	//
	//	List of READ (and WRITE) commands.
	// NOTE: Monitoring loop stops on first cmd = ''.
	//
	cmdList_Read_HIPACE30:	ARRAY [1..16] OF T_CRYO_PUMP_CMD := [
		(cmd := cfg.C_CMD_bON, 				length := 20),	// 20 chars with the terminator!	
		(cmd := cfg.C_CMD_nCtrlMode, 		length := 17),	
		(cmd := cfg.C_CMD_sErrorCode, 		length := 20),
		(cmd := cfg.C_CMD_bTargetSpeed, 	length := 20),
		(cmd := cfg.C_CMD_nMotorCurr, 		length := 20),
		(cmd := cfg.C_CMD_nPumpHours, 		length := 20),
		(cmd := cfg.C_CMD_nMotorVolt, 		length := 20),
		(cmd := cfg.C_CMD_nElecHours, 		length := 20),
		(cmd := cfg.C_CMD_nElecTemp, 		length := 20),
		(cmd := cfg.C_CMD_nPumpTemp, 		length := 20),
		(cmd := cfg.C_CMD_nPumpSpeed, 		length := 20),
		(cmd := '', 						length := 0),
		(cmd := '', 						length := 0),
		(cmd := '', 						length := 0),
		(cmd := '', 						length := 0),
		(cmd := '', 						length := 0)];
	
		i:	INT;
END_VAR
IF NOT bStarted	THEN
	//
	// START: Mandatory for ALL pumps !!!
	//
	// Set references from FB_RS_BASE
	cfgRef	REF=cfg;
	ctrlRef	REF=ctrl;
	statRef	REF=stat;

	// Set references from FB_CRYO_TMP_BASE
	cfgBaseRef	REF=cfg;
	ctrlBaseRef	REF=ctrl;
	statBaseRef	REF=stat;
	
	// Copy input parameters to configuration
	cfg.nModel			:= in_nModel;
	cfg.bAutoMonitor	:= in_bAutoMonitor;
	cfg.tDelay_Periodic	:= DINT_TO_TIME(in_nPeriod);
	
	
	// Set pointers to arrays of commands
	ptrInitCmds	:= ADR(cfg.cmdList_Init);(* Pointer to INIT commands *)
	ptrReadCmds	:= ADR(cfg.cmdList_Read);(* Pointer to READ commands *)
	
	// TODO in FB that extends the functionality
	// Set pointers to comm, i.e.
	ptrCommCfg	:= ADR(comm.cfg);	(* Pointer to comm.cfg instance *)
	ptrCommCtrl	:= ADR(comm.ctrl);	(* Pointer to comm.ctrl instance *)
	ptrCommStat	:= ADR(comm.stat);	(* Pointer to comm.stat instance *)
	
	// Set comm suffixes for commands and replies
	ptrCommCfg^.sCmdSuffix		:= in_sCmdSuffix;
	ptrCommCfg^.sReplySuffix	:= in_sReplySuffix;

	statRef.bConfigured	:= TRUE;
	bStarted			:= TRUE;
	//
	// END: Mandatory for ALL pumps !!!
	//


	//
	// ATH specific configuration
	//
	
	// Assign INIT and READ commands.
	cfg.cmdList_Init	:= cmdList_Init_HIPACE30;
	cfg.cmdList_Read	:= cmdList_Read_HIPACE30;
	
	// Add checksum to all INIT and READ commands
	FOR i:=1 TO 8 DO
		IF cfg.cmdList_Init[i].cmd <> '' THEN
			cfg.cmdList_Init[i].cmd	:= M_PVP_Checksum(cfg.cmdList_Init[i].cmd);
		ELSE
			EXIT;
		END_IF
	END_FOR
	
	FOR i:=1 TO 16 DO
		IF cfg.cmdList_Read[i].cmd <> '' THEN
			cfg.cmdList_Read[i].cmd	:= M_PVP_Checksum(cfg.cmdList_Read[i].cmd);
		ELSE
			EXIT;
		END_IF
	END_FOR
	
END_IF
END_METHOD

METHOD M_GetSpeed : DINT
VAR_INPUT
END_VAR
M_GetSpeed	:= stat.nPumpSpeed;
END_METHOD

METHOD M_IsReady : BOOL
VAR_INPUT
END_VAR
M_IsReady	:= stat.bReady;
END_METHOD

METHOD M_IsRunning : BOOL
VAR_INPUT
END_VAR
M_IsRunning	:= stat.bMoving;
END_METHOD

METHOD M_ReadFromReply : BOOL
// Method to check correctness of the reply and assign the result to a status variable.
VAR_INPUT
	idx:		INT;		(* arr [idx] will hold the first extracted value, arr [idx+1] the second one, etc. *)
	bInitCmd:	BOOL := FALSE;
END_VAR
VAR
	pos:	INT;
	cmd:	STRING;
	length:	DINT;
	subStr:	STRING;
	valLen:	INT;		// Number of character for the value
END_VAR
// During INIT it might happen that the command index is 0.
// These cases should be discarded.
IF idx <= 0	THEN
	M_ReadFromReply	:= TRUE;
	RETURN;
END_IF

IF bInitCmd	THEN
	cmd		:= cfg.cmdList_Init[idx].cmd;
	length	:= cfg.cmdList_Init[idx].length;
ELSE
	cmd		:= cfg.cmdList_Read[idx].cmd;
	length	:= cfg.cmdList_Read[idx].length;
END_IF

IF length <> 0  AND  LEN(stat.sReply) <> length THEN
	stat.sErrorText	:= 'Wrong reply length';
	M_ReadFromReply	:= FALSE;
	RETURN;
END_IF

// Check if sent command was correct.
IF	FIND(stat.sReply,'NO_DEF') > 0	OR 
	FIND(stat.sReply,'_RANGE') > 0	OR 
	FIND(stat.sReply,'_LOGIC') > 0		THEN
	// Wrong command sent. This is an error.
	stat.sErrorText	:= 'Incorrect command';
	M_ReadFromReply	:= FALSE;
	RETURN;
END_IF

// Check the structure of the reply.
// Example 1 - Data query with 6 characters for the value:
//    CMD:   1 2 3 0 0 3 0 9 0 2 = ? 1 1 2 cR
//    Reply: 1 2 3 1 0 3 0 9 0 6 0 0 0 6 3 3 0 3 7 cR
//    valLen = 6 (from '06' in reply)
//    value = 633
// Example 2 - Data query with 3 characters for the value:
//    CMD:   1 2 3 0 0 0 6 0 0 2 = ? x x x cR
//    Reply: 1 2 3 1 0 0 6 0 0 3 0 0 2 y y y cR
//    valLen = 3 (from '03' in reply)
//    value = 002 = 2
// Example 3 - Command (reply is identical to command):
//    CMD:   0 4 2 1 0 0 1 0 0 6 1 1 1 1 1 1 0 2 0 cR
//    Reply: 0 4 2 1 0 0 1 0 0 6 1 1 1 1 1 1 0 2 0 cR
//    valLen = 6 (from '06' in reply)
//    value = 111111
//
// Compared to the first 10 chars of the command, 
// the reply should modify characters 3 and 9 (index starts from 0)
// reply[3] = 1
// reply[9] = length - 14
//
// So, we want to convert: 1 2 3 0 0 3 0 9 0 2
//                     to: 1 2 3 1 0 3 0 9 0 6
// Extract first 10 characters from the command
subStr	:= MID(cmd,10,1);
// Replace character [3] with '1', i.e. with ASCII 49.
subStr[3]	:= 49;
// Replace character [9] with expected number of characters in the value.
valLen	:= DINT_TO_INT(length - 14);
// Convert integer to character.
subStr[9]	:= INT_TO_BYTE(valLen + 48);	// 48 is ascii '0'.
IF	FIND(stat.sReply,subStr) <> 1	THEN
	// Wrong reply received. This is an error.
	stat.sErrorText	:= 'Wrong reply received';
	M_ReadFromReply	:= FALSE;
	RETURN;
END_IF


//
// All fine so far. Let's extract the reading.
//
// The actual reply is contained in the 'valLen' (3 or 6) characters starting 
// from char [10] (11-the character for MID() function).
subStr	:= MID(stat.sReply, valLen, 11);

// Remove the 3-character checksum from the command.
cmd	:= MID(cmd, LEN(cmd)-3,1);


IF cmd = cfg.C_CMD_sFwVersion	THEN
	stat.sFwVersion		:= MID(subStr, 6, 1);
ELSIF cmd = cfg.C_CMD_sHwVersion	THEN
	stat.sHwVersion		:= MID(subStr, 6, 1);
ELSIF cmd = cfg.C_CMD_nNominalSpeed	THEN
	stat.nNominalSpeed	:= LREAL_TO_DINT(STRING_TO_LREAL(subStr));
ELSIF cmd = cfg.C_CMD_bON	THEN
	stat.bON	:= STRING_TO_BOOL(subStr) <> FALSE;
ELSIF cmd = cfg.C_CMD_nCtrlMode	THEN
	stat.nCtrlMode	:= STRING_TO_DINT(subStr);
ELSIF cmd = cfg.C_CMD_sErrorCode	THEN
	IF	FIND(subStr,'Err') > 0	OR 
		FIND(subStr,'Wrn') > 0		THEN
		// There is an Error or Warning.
		stat.sFailureCode	:= MID(subStr, 6, 1);
		stat.bFailure		:= TRUE;
	ELSE
		stat.sFailureCode	:= 'OK';
		stat.bFailure		:= FALSE;
	END_IF
ELSIF cmd = cfg.C_CMD_bTargetSpeed	THEN
	stat.bTargetSpeed	:= STRING_TO_BOOL(subStr) <> FALSE;
ELSIF cmd = cfg.C_CMD_nMotorCurr	THEN
	stat.nMotorCurr	:= STRING_TO_DINT(subStr) * 10;	// [mA]
ELSIF cmd = cfg.C_CMD_nPumpHours	THEN
	stat.nPumpHours	:= STRING_TO_DINT(subStr);
ELSIF cmd = cfg.C_CMD_nMotorVolt	THEN
	stat.nMotorVolt	:= STRING_TO_DINT(subStr) / 100;
	stat.lrMotorVolt:= STRING_TO_LREAL(subStr) / 100.0;	// [V]
ELSIF cmd = cfg.C_CMD_nElecHours	THEN
	stat.nElecHours	:= STRING_TO_DINT(subStr);
ELSIF cmd = cfg.C_CMD_nElecTemp	THEN
	stat.nElecTemp	:= STRING_TO_DINT(subStr);
ELSIF cmd = cfg.C_CMD_nPumpTemp	THEN
	stat.nPumpTemp	:= STRING_TO_DINT(subStr);
ELSIF cmd = cfg.C_CMD_nPumpSpeed	THEN
	stat.nPumpSpeed	:= LREAL_TO_DINT(STRING_TO_LREAL(subStr));
END_IF


M_ReadFromReply	:= TRUE;	// OK
END_METHOD

METHOD M_UpdateStatus
VAR_INPUT
END_VAR
// Update Status from digital inputs readings
stat.bReady		:= i_bReady;
stat.bFailure	:= NOT i_bError;	// Active low

stat.bMoving	:= stat.bReady OR stat.nPumpSpeed > 0;

// Set Control Mode Label
(*
	1 = remote
	2 = RS-485
	4 = PV.can
	8 = Fieldbus
	16 = E74
	255 = unlock interface selection
*)
CASE stat.nCtrlMode	OF
	1:		stat.sCtrlMode	:= 'REMOTE';
	2:		stat.sCtrlMode	:= 'RS-485';
	4:		stat.sCtrlMode	:= 'PV.can';
	8:		stat.sCtrlMode	:= 'FIELDBUS';
	16:		stat.sCtrlMode	:= 'E74';
ELSE
	stat.sCtrlMode	:= 'UNKNOWN';
END_CASE
END_METHOD

END_FUNCTION_BLOCK

// ---- POUs/Subsystems/Examples/Evacuation/FB_CRYO_EVAC_ECODRY_ATH2303M.TcPOU
FUNCTION_BLOCK FB_CRYO_EVAC_ECODRY_ATH2303M EXTENDS FB_CRYO_EVAC_BASE
VAR_INPUT
END_VAR
VAR_OUTPUT
END_VAR
VAR
	rp:	FB_CRYO_PUMP_ECODRY;	// Roughing Pump
	tp:	FB_CRYO_PUMP_ATH2303M;	// Turbo Molecular Pump
	
END_VAR

SUPER^();

METHOD M_Configure
VAR_INPUT
END_VAR
//
// Specific PDS IR Imager configuration.
//
IF NOT stat.bConfigured	THEN
	// MANDATORY: Set References !!!
	// If not done, system will crash !!!
	rpRef	REF=rp;
	tpRef	REF=tp;
	

	// Specific instance configuration, e.g. anything different
	// from the default values given in the cfg structure of type T_CRYO_EVAC_CFG.
	cfg.nPressGaugeType1	:= E_CRYO_SENSOR_TYPE_PRESS.WRG_D_NW25;
	cfg.nPressGaugeType2	:= E_CRYO_SENSOR_TYPE_PRESS.PKR_360;

	cfg.lrThld_Prevac := 5.0;	// Prevacuum pressure threshold
	// Cryo pressure threshold to start Turbo Pump before opening Valve
	cfg.lrThld_TP_SafeStartPressure := 0.01;	
	// Cryo pressure threshold to start Turbo Pump once Valve is open
	cfg.lrThld_Valve_SafeOpenPressure := 0.1;	
	cfg.tDelay := T#3S;	// Time delay before stopping Turbo Pump

	stat.bConfigured	:= TRUE;;
ELSE
	RETURN;	// Nothing to do any more
END_IF
END_METHOD

METHOD M_ExecuteControllers
VAR_INPUT
END_VAR
//
// Specific Cryo Lab Evacuation System HW configuration.
//

// Roughing Pump	
rp(	
	in_bSimulation	:= FALSE,
	in_sName		:= 'ECODRY V01',
	in_bEnable		:= ctrl.bEnable_RP,
	in_nSlaveID		:= 31,
	in_sVersion		:= 'V01',
	in_nPeriod		:= 2000);

// Turbo Molecular Pump
tp(	
	in_bSimulation	:= FALSE,
	in_sName		:= 'ATH2303M',
	in_bEnable		:= ctrl.bEnable_TP,
	in_nModel		:= 2303,
	in_bAutoMonitor	:= TRUE,
	in_nPeriod		:= 2000);

// Valve
valve(
	in_bEnable		:= ctrl.bEnable_Valve,
	in_nFeedback	:= E_CRYO_BIN_ACT_FEEDBACK.ON_AND_OFF);
END_METHOD

END_FUNCTION_BLOCK

// ---- POUs/Pumps/FB_CRYO_PUMP_ECODRY.TcPOU
FUNCTION_BLOCK FB_CRYO_PUMP_ECODRY EXTENDS FB_CRYO_PUMP_MODBUS
VAR_INPUT
END_VAR
VAR_OUTPUT
END_VAR
VAR CONSTANT
END_VAR
VAR
	{attribute 'OPC.UA.DA' := '1'}
	cfg:		T_CRYO_PUMP_MODBUS_CFG;		//  Config parameters
	{attribute 'OPC.UA.DA' := '1'}
	ctrl:		T_CRYO_PUMP_MODBUS_CTRL;	//  Control parameters
	{attribute 'OPC.UA.DA' := '1'}
	{attribute 'OPC.UA.DA.Access' := '1'}
	stat:		T_CRYO_PUMP_MODBUS_STAT;	//  Status parameters - ReadOnly


END_VAR

// Execute the base class object FB_RS_BASE
SUPER^();

METHOD M_Configure
VAR_INPUT
END_VAR
IF NOT bStarted	THEN
	//
	// START: Mandatory for ALL pumps !!!
	//
	// Set references from FB_RS_BASE
	cfgRef	REF=cfg;
	ctrlRef	REF=ctrl;
	statRef	REF=stat;

	// Set references from FB_CRYO_PUMP_BASE
	cfgBaseRef	REF=cfg;
	ctrlBaseRef	REF=ctrl;
	statBaseRef	REF=stat;

	// Set references from FB_CRYO_PUMP_MODBUS
	cfgModbusRef	REF=cfg;
	ctrlModbusRef	REF=ctrl;
	statModbusRef	REF=stat;

	// Copy input parameters to configuration
	cfg.nModel			:= in_nModel;
	cfg.bAutoMonitor	:= in_bAutoMonitor;
	cfg.tDelay_Periodic	:= DINT_TO_TIME(in_nPeriod);
	
	
	// Set pointers to arrays of commands
//	ptrInitCmds	:= ADR(cfg.cmdList_Init);(* Pointer to INIT commands *)
//	ptrReadCmds	:= ADR(cfg.cmdList_Read);(* Pointer to READ commands *)
	
	// TODO in FB that extends the functionality
	// Set pointers to comm, i.e.
	ptrCommCfg	:= ADR(comm.cfg);	(* Pointer to comm.cfg instance *)
	ptrCommCtrl	:= ADR(comm.ctrl);	(* Pointer to comm.ctrl instance *)
	ptrCommStat	:= ADR(comm.stat);	(* Pointer to comm.stat instance *)
	
	// Set comm suffixes for commands and replies
//	ptrCommCfg^.sCmdSuffix		:= '';
//	ptrCommCfg^.sReplySuffix	:= '';

	statRef.bConfigured	:= TRUE;
	bStarted			:= TRUE;
	//
	// END: Mandatory for ALL pumps !!!
	//


	// TODO USER
	// Add here real configuration
	IF in_sVersion = 'V01'	THEN
		cfg.nVersion	:= E_ECODRY_VERSION.V01;
	ELSIF in_sVersion = 'V21'  OR  in_sVersion = 'V22'	THEN
		cfg.nVersion	:= E_ECODRY_VERSION.V21_22;
	END_IF
	
	// Adjust addresses and number of words
	CASE cfg.nVersion	OF
		E_ECODRY_VERSION.V01:
			// Set register addresses
			cfg.aAddr [1]	:= 16#0040;
			cfg.aAddr [2]	:= 16#0067;
			cfg.aAddr [3]	:= 16#0667;
			cfg.aAddr [4]	:= 0;	// Unused address must be zero
			
			// Set number of words to read
			cfg.aWords [1]	:= 16;
			cfg.aWords [2]	:= 2;
			cfg.aWords [3]	:= 6;
			cfg.aWords [4]	:= 0;	// Number of words for unused address must be zero
	END_CASE
	
	cfg.nSlaveID	:= in_nSlaveID;

	
END_IF
END_METHOD

METHOD M_ExtractReadings_V01 : BOOL
VAR_INPUT
	nAddressIndex:	INT;	// Which address space to read
END_VAR
VAR
	pBuf:	POINTER TO BYTE	:= ADR(stat.nInputBuffer);
	loop:	INT;
	par:	INT;
END_VAR
// There are 3 bytes before data starts !!!
IF nAddressIndex = 1 THEN
	////////////////////////////
	// Extract Common Parameters
	////////////////////////////

	// Reference Frequency 0x40H
	// Offset 3 + 0 = 3
	stat.lrFreqRef		:= UINT_TO_LREAL(M_ByteSwapUINT(ADR(pBuf[3]))) / 100.0;
	stat.lrOutFreq		:= INT_TO_LREAL(M_ByteSwapINT(ADR(pBuf[5]))) / 100.0;
	stat.nPumpSpeed		:= LREAL_TO_DINT(stat.lrOutFreq * 60.0);	// [Hz] -> [rpm]
	stat.nMotorCurr		:= UINT_TO_DINT(M_ByteSwapUINT(ADR(pBuf[7]))) * 10;
	stat.lrOutVoltRef	:= UINT_TO_LREAL(M_ByteSwapUINT(ADR(pBuf[13]))) / 10.0;
	stat.nMotorVolt		:= UINT_TO_DINT(M_ByteSwapUINT(ADR(pBuf[15])));
	stat.lrOutPower		:= INT_TO_LREAL(M_ByteSwapINT(ADR(pBuf[17]))) / 10.0;
	
	stat.nOpTime	:= M_ByteSwapUINT(ADR(pBuf[27]));
	stat.nSwFlash	:= M_ByteSwapUINT(ADR(pBuf[29]));

	(*
	stat.lrTemperature	:= UINT_TO_LREAL(M_ByteSwapUINT(ADR(pBuf[83])));

	stat.nSwRom		:= M_ByteSwapUINT(ADR(pBuf[57]));
	stat.nNumRunCmd	:= M_ByteSwapUINT(ADR(pBuf[109]));
	stat.nFanOpTime	:= M_ByteSwapUINT(ADR(pBuf[81]));
	*)

ELSIF nAddressIndex = 2 THEN
	stat.nFanOpTime			:= M_ByteSwapUINT(ADR(pBuf[3]));
	stat.nElecTemp			:= UINT_TO_DINT(M_ByteSwapUINT(ADR(pBuf[5])));
ELSIF nAddressIndex = 3 THEN
	stat.nServiceHours		:= M_ByteSwapUINT(ADR(pBuf[3]));
	stat.nNumPumpDowns		:= M_ByteSwapUINT(ADR(pBuf[7]));
	stat.nDaysUntilService	:= M_ByteSwapUINT(ADR(pBuf[13]));
END_IF
END_METHOD

METHOD M_ExtractReadings_V21_22 : BOOL
VAR_INPUT
	nAddressIndex:	INT;	// Which address space to read
END_VAR
VAR
	pBuf:	POINTER TO BYTE	:= ADR(stat.nInputBuffer);
	loop:	INT;
	par:	INT;
END_VAR
// There are 3 bytes before data starts !!!
IF nAddressIndex = 1 THEN
	////////////////////////////
	// Extract Common Parameters
	////////////////////////////

	// Reference Frequency 0x40H
	// Offset 3 + 0 = 3
	stat.lrFreqRef		:= UINT_TO_LREAL(M_ByteSwapUINT(ADR(pBuf[3]))) / 100.0;
	stat.lrOutFreq		:= INT_TO_LREAL(M_ByteSwapINT(ADR(pBuf[5]))) / 100.0;
	stat.nMotorCurr		:= UINT_TO_DINT(M_ByteSwapUINT(ADR(pBuf[7]))) * 10;
	stat.lrOutVoltRef	:= UINT_TO_LREAL(M_ByteSwapUINT(ADR(pBuf[13]))) / 10.0;
	stat.nMotorVolt		:= UINT_TO_DINT(M_ByteSwapUINT(ADR(pBuf[15])));
	stat.lrOutPower		:= INT_TO_LREAL(M_ByteSwapINT(ADR(pBuf[17]))) / 10.0;
	
	stat.nOpTime	:= M_ByteSwapUINT(ADR(pBuf[27]));
	stat.nSwFlash	:= M_ByteSwapUINT(ADR(pBuf[29]));

	(*
	stat.lrTemperature	:= UINT_TO_LREAL(M_ByteSwapUINT(ADR(pBuf[83])));

	stat.nSwRom		:= M_ByteSwapUINT(ADR(pBuf[57]));
	stat.nNumRunCmd	:= M_ByteSwapUINT(ADR(pBuf[109]));
	stat.nFanOpTime	:= M_ByteSwapUINT(ADR(pBuf[81]));
	*)

ELSIF nAddressIndex = 2 THEN
	stat.nFanOpTime			:= M_ByteSwapUINT(ADR(pBuf[3]));
	stat.nElecTemp			:= UINT_TO_DINT(M_ByteSwapUINT(ADR(pBuf[5])));
ELSIF nAddressIndex = 3 THEN
	stat.nServiceHours		:= M_ByteSwapUINT(ADR(pBuf[3]));
	stat.nNumPumpDowns		:= M_ByteSwapUINT(ADR(pBuf[7]));
	stat.nDaysUntilService	:= M_ByteSwapUINT(ADR(pBuf[13]));
END_IF
END_METHOD

METHOD M_IsReady : BOOL
VAR_INPUT
END_VAR
//	M_UpdateStatus() sets the stat.bReady flag.
M_IsReady	:= stat.bReady;
END_METHOD

METHOD M_IsRunning : BOOL
VAR_INPUT
END_VAR
M_IsRunning	:= stat.bReady OR stat.nPumpSpeed > 0;
END_METHOD

METHOD M_ReadFromReply : BOOL
VAR_INPUT
	nAddressIndex:	INT;	// Which address space to read
END_VAR
IF cfg.nVersion	= E_ECODRY_VERSION.V01	THEN
	M_ExtractReadings_V01    (nAddressIndex);
ELSIF cfg.nVersion	= E_ECODRY_VERSION.V21_22	THEN
	M_ExtractReadings_V21_22 (nAddressIndex);
END_IF
END_METHOD

METHOD M_UpdateStatus
VAR_INPUT
END_VAR
// Update inputs
stat.bReady		:= NOT i_bRunning;	// Active low
END_METHOD

END_FUNCTION_BLOCK

// ---- POUs/Pumps/FB_CRYO_PUMP_MODBUS.TcPOU
FUNCTION_BLOCK FB_CRYO_PUMP_MODBUS EXTENDS FB_CRYO_PUMP_BASE
VAR_INPUT
	{attribute 'OPC.UA.DA' := '0'}
	in_nSlaveID:	BYTE := 1;		// Slave ID
	{attribute 'OPC.UA.DA' := '0'}
	in_sVersion:	STRING := 'V21';	// Version number. String starting with 'V', e.g. 'V21'.
END_VAR
VAR_OUTPUT
END_VAR
VAR CONSTANT
END_VAR
VAR
	{attribute 'OPC.UA.DA' := '0'}
	cfgModbusRef:	REFERENCE TO T_CRYO_PUMP_MODBUS_CFG;
	{attribute 'OPC.UA.DA' := '0'}
	ctrlModbusRef:	REFERENCE TO T_CRYO_PUMP_MODBUS_CTRL;
	{attribute 'OPC.UA.DA' := '0'}
	statModbusRef:	REFERENCE TO T_CRYO_PUMP_MODBUS_STAT;
	
	{attribute 'OPC.UA.DA' := '0'}
	comm:		FB_MODBUS_COMM_NO_SIM;		// Instance of generic comm object. OPC UA Disabled!!!
	
	(* Pointers *)
	{attribute 'OPC.UA.DA' := '0'}
	ptrCommCfg:		POINTER TO T_MODBUS_CFG 	:= ADR(comm.cfg);	(* Pointer to comm.cfg instance *)
	{attribute 'OPC.UA.DA' := '0'}
	ptrCommCtrl:	POINTER TO T_MODBUS_CTRL 	:= ADR(comm.ctrl);	(* Pointer to comm.ctrl instance *)
	{attribute 'OPC.UA.DA' := '0'}
	ptrCommStat:	POINTER TO T_MODBUS_STAT 	:= ADR(comm.stat);	(* Pointer to comm.stat instance *)


	(* Timers *)


	// Input signals
	i_bRunning		AT %I*:	BOOL;	// TRUE, if pump is running


END_VAR

// Execute the base class object FB_CRYO_PUMP_BASE
SUPER^();

METHOD ActivityInitializing
VAR_INPUT
	bExecute:	BOOL;
END_VAR
VAR_INST
	{attribute 'OPC.UA.DA' := '0'}
    nMethodState:	INT := 0;	// State Machine current state
END_VAR
VAR
	nInt:	INT;	// Temporary INT for conversion of ENUM types
END_VAR
SetAction('ActivityInitializing');


IF NOT bExecute THEN
	nMethodState	:= 0;	// Reset the state machine
	RETURN;
END_IF

// Handle State Machine
CASE nMethodState OF
	0:	// Set communication parameters and Model configuration


		// Set monitoring period (input parameter)
		cfgRef.tDelay_Periodic	:= DINT_TO_TIME(in_nPeriod);
		// Auto monitor, i.e. monitor in Standby_Ready as well
		cfgRef.bAutoMonitor	:= TRUE;

		(* Set initial state and status *)
		statRef.bInitialised	:= FALSE;
		statBaseRef.nRetries		:= 0;

		SetStatus(E_SM_ERROR.OK, 'BUSY');
		
		// User configuration of the system
//		M_UserConfigure();

		nMethodState := 10;				// Go to next state, i.e. INIT_COMM

	10:	// Initialize COMM port
		(* Reset the serial port *)
		nInt	:= E_RS_COMM_CMD.INIT;
		ptrCommCtrl^.nCommand	:= nInt;
		ptrCommCtrl^.bExecute	:= TRUE;

		(* Start the timer by going false/true *)
		fbTimer (IN := FALSE); (* Reset timer *)
		fbTimer (IN := TRUE, PT := T#5S); (* 5 sec timeout for reply *)

		nMethodState 	:= 15;	// On next cycle wait until the comm port is reset, i.e. idle
		
	15:	// Wait IDLE
		fbTimer (IN := TRUE);
		IF comm.stat.nStatus = E_RS_COMM_STATUS.IDLE THEN
			// Communication is IDLE 
			fbTimer (IN := FALSE);	// disable timer 
			statModbusRef.nInputBuffer		:= ptrCommStat^.DeviceReply;	// Save the reply

			bCommProblem	:= FALSE;
			// Device INIT is done. Go to IDLE 
			statRef.bInitialised 	:= TRUE;
			SetStatus(E_CCC_STATUS.IDLE, 'IDLE');
			nEvent 		:= E_SM_EVENT.INITDONE;
			RETURN;
		ELSIF comm.stat.nStatus = E_RS_COMM_STATUS.ERROR THEN
			fbTimer (IN := FALSE);
			SetStatus(E_CCC_ERROR.COMM, 'ERROR: Communication error');	
			bCommProblem	:= TRUE;
			nEvent := E_SM_EVENT.ERRINIT;
			RETURN;
		ELSIF fbTimer.Q THEN
			// Timer expired after 5 sec. This is an error.
			fbTimer (IN := FALSE);
			SetStatus(E_CCC_ERROR.TIMEOUT, 'ERROR: Communication timeout');	
			bCommProblem	:= TRUE;
			nEvent := E_SM_EVENT.ERRINIT;
			RETURN;
		END_IF

	
	
	
END_CASE
END_METHOD

METHOD ActivityMonitoring
VAR_INPUT
	bExecute:	BOOL;
END_VAR
VAR_INST
	{attribute 'OPC.UA.DA' := '0'}
    nMethodState:	INT := 0;			// State Machine current state
	{attribute 'OPC.UA.DA' := '0'}
	nAddressIndex:	INT := 1;			// Which address space to read
	{attribute 'OPC.UA.DA' := '0'}
	nRetries:		INT := 0;			// Number of retries in case of communication problems
END_VAR
IF NOT bExecute THEN
	SetAction('ActivityMonitoring'); 
	SetStatus(E_SM_ERROR.OK, 'BUSY');
	nMethodState	:= 0;	// Reset the state machine
	nAddressIndex	:= 1;
	ctrlModbusRef.nRegister	:= cfgModbusRef.aAddr  [1];
	ctrlModbusRef.nWords	:= cfgModbusRef.aWords [1];
	nRetries		:= 0;					
	RETURN;
END_IF

// Handle State Machine
CASE nMethodState OF
	0:	// Execute a command from the command array
		// Check if we have to exit Monitoring
		IF nNextState <> E_RS_BASE_STATE.NONE	THEN
			SetStatus(E_SM_ERROR.OK, nNextDescription);
			SetState(nNextState, nNextSubstate);
			nNextState		:= E_RS_BASE_STATE.NONE;
			nNextSubstate	:= E_RS_BASE_SUBSTATE.NONE;
			nNextDescription:= 'IDLE';
			RETURN;
		END_IF
		
		
		// Send command
		ptrCommCtrl^.nCommand		:= E_MODBUS_CMD.SEND;
		ptrCommCtrl^.nSlaveID		:= cfgModbusRef.nSlaveID;
		ptrCommCtrl^.nRegister		:= ctrlModbusRef.nRegister;
		ptrCommCtrl^.nWords			:= ctrlModbusRef.nWords;
		ptrCommCtrl^.bExecute		:= TRUE;
		
		(* Start the timer by going false/true *)
		fbTimer (IN := FALSE); (* Reset timer *)
		fbTimer (IN := TRUE, PT := T#5S); (* 5 sec timeout for reply *)

		nMethodState := 20;				// Goto WAIT for Reading to complete,

	10:	// Wait until the delay timeout expires
		fbTimer (IN := TRUE);

		// Check if we have to exit Monitoring
		IF nNextState <> E_RS_BASE_STATE.NONE THEN
			fbTimer (IN := FALSE); (* Stop the timer *)
			SetStatus(E_SM_ERROR.OK, nNextDescription);
			SetState(nNextState, nNextSubstate);
			nNextState		:= E_RS_BASE_STATE.NONE;
			nNextSubstate	:= E_RS_BASE_SUBSTATE.NONE;
			nNextDescription:= 'IDLE';
			RETURN;
		END_IF
	
		(* If Timer has expired, go to the next state. *)
		IF fbTimer.Q THEN
			fbTimer (IN := FALSE);
			SetStatus(E_SM_ERROR.OK, 'BUSY');
			nMethodState 	:= 0;	// Goto next reading
			RETURN;
		END_IF
	


	20:	// Wait for the reading to complete, i.e. IDLE
		fbTimer (IN := TRUE);
		IF comm.stat.nStatus = E_RS_COMM_STATUS.IDLE THEN
			// Communication is IDLE  
			fbTimer (IN := FALSE);	// disable timer 
			statModbusRef.nInputBuffer		:= ptrCommStat^.DeviceReply;	// Save the reply
			
			// Extract the readings from the reply.
			M_ReadFromReply(nAddressIndex);

			bCommProblem	:= FALSE;
			nRetries		:= 0;	// Reset number of retries
			
			// Check if we have to exit Monitoring
			IF nNextState <> E_RS_BASE_STATE.NONE THEN
				fbTimer (IN := FALSE); (* Stop the timer *)
				SetStatus(E_SM_ERROR.OK, nNextDescription);
				SetState(nNextState, nNextSubstate);
				nNextState		:= E_RS_BASE_STATE.NONE;
				nNextSubstate	:= E_RS_BASE_SUBSTATE.NONE;
				nNextDescription:= 'IDLE';
				RETURN;
			END_IF
	
			IF NOT M_SetCommand(nAddressIndex) THEN
				// We completed a full read cycle.
				// Wait periodic delay.
				// Periodic READ is done. Wait tDelay_Periodic before re-starting the READ.
				SetStatus(E_SM_ERROR.OK, 'IDLE');
				(* Start the timer by going false/true *)
				fbTimer (IN := FALSE); (* Reset timer *)
				fbTimer (IN := TRUE, PT := cfgRef.tDelay_Periodic);
				nMethodState := 10;				// Goto Wait 
				RETURN;
			ELSE
				// Apply a short delay of 30 ms after each command
				fbTimer (IN := FALSE); (* Reset timer *)
				fbTimer (IN := TRUE, PT := T#30MS);
				nMethodState := 10;				// Goto Wait 
				RETURN;
			END_IF

		ELSIF INT_TO_DINT(comm.stat.nStatus) = INT_TO_DINT(E_MODBUS_STATUS.ERROR) OR fbTimer.Q THEN
			fbTimer (IN := FALSE);
			SetStatus(E_MODBUS_ERROR.RECEIVE, 'ERROR: Communication error');	
			bCommProblem	:= TRUE;
			// Retry up to 3 times
			nRetries		:= nRetries + 1;		// Increment number of retries
			statModbusRef.nRetries	:= statModbusRef.nRetries + 1;	// Increment total number of retries
			IF nRetries > 3 THEN
				nEvent := E_SM_EVENT.ERRCOMM;
			ELSE
				// Apply a short delay of 1 sec and retry
				fbTimer (IN := FALSE); (* Reset timer *)
				fbTimer (IN := TRUE, PT := T#1000MS);
				nMethodState := 10;				// Goto Wait 
			END_IF
			RETURN;
		END_IF

	
END_CASE
END_METHOD

METHOD M_ByteSwapFLOAT : REAL
VAR_INPUT
	pByte:		POINTER TO BYTE;	// Pointer to array of bytes read from JUMO
END_VAR
VAR
	rResult:	REAL;
	pResult:	POINTER TO BYTE	:= ADR(rResult);	// Pointer to the result
END_VAR
pResult[0]	:= pByte[1];
pResult[1]	:= pByte[0];
pResult[2]	:= pByte[3];
pResult[3]	:= pByte[2];

M_ByteSwapFLOAT	:= rResult;
END_METHOD

METHOD M_ByteSwapINT : INT
VAR_INPUT
	pByte:		POINTER TO BYTE;	// Pointer to array of bytes read from JUMO
END_VAR
VAR
	nResult:	INT;
	pResult:	POINTER TO BYTE	:= ADR(nResult);	// Pointer to the result
END_VAR
pResult[0]	:= pByte[1];
pResult[1]	:= pByte[0];

M_ByteSwapINT	:= nResult;
END_METHOD

METHOD M_ByteSwapUINT : UINT
VAR_INPUT
	pByte:		POINTER TO BYTE;	// Pointer to array of bytes read from JUMO
END_VAR
VAR
	nResult:	UINT;
	pResult:	POINTER TO BYTE	:= ADR(nResult);	// Pointer to the result
END_VAR
pResult[0]	:= pByte[1];
pResult[1]	:= pByte[0];

M_ByteSwapUINT	:= nResult;
END_METHOD

METHOD M_ExecuteComm
VAR_INPUT
END_VAR
(* Execute comm instance *)
comm(	in_bSimulation	:= in_bSimulation,
		in_nModel		:= 0,
		in_cReadFunction:= 3);
END_METHOD

METHOD M_GetCouplerState : BOOL
VAR_INPUT
END_VAR
IF comm.i_nCouplerState = 8 THEN
	M_GetCouplerState	:= TRUE;	
ELSE
	M_GetCouplerState	:= FALSE;	
END_IF
END_METHOD

METHOD M_ReadFromReply : BOOL
VAR_INPUT
	nAddressIndex:	INT;	// Which address space to read
END_VAR
// TODO: For every pump implementation
END_METHOD

METHOD M_SetCommand : BOOL
VAR_IN_OUT
	nAddressIndex:	INT;	// Which address space to read
END_VAR
// We always read from ECODRY
ctrlModbusRef.nCmdType	:= E_MODBUS_CMD_TYPE.READ;

// Go to next register address to read
nAddressIndex	:= nAddressIndex + 1;

IF nAddressIndex > 8  OR  cfgModbusRef.aAddr[nAddressIndex] = 0	OR  cfgModbusRef.aWords[nAddressIndex] = 0	THEN
	ctrlModbusRef.nRegister	:= cfgModbusRef.aAddr  [1];
	ctrlModbusRef.nWords	:= cfgModbusRef.aWords [1];
	nAddressIndex	:= 1;
	M_SetCommand	:= FALSE;	// Restarting from first address
ELSE
	ctrlModbusRef.nRegister	:= cfgModbusRef.aAddr  [nAddressIndex];
	ctrlModbusRef.nWords	:= cfgModbusRef.aWords [nAddressIndex];
	M_SetCommand	:= TRUE;	
END_IF
END_METHOD

END_FUNCTION_BLOCK

// ---- POUs/Pumps/FB_CRYO_PUMP_ATH2303M.TcPOU
FUNCTION_BLOCK FB_CRYO_PUMP_ATH2303M EXTENDS FB_CRYO_PUMP_SERIAL
VAR_INPUT
END_VAR
VAR_OUTPUT
END_VAR
VAR
	{attribute 'OPC.UA.DA' := '1'}
	cfg:		T_CRYO_PUMP_ATM2303M_CFG;	
	{attribute 'OPC.UA.DA' := '1'}
	ctrl:		T_CRYO_PUMP_BASE_CTRL;	
	{attribute 'OPC.UA.DA' := '1'}
	{attribute 'OPC.UA.DA.Access' := '1'}
	stat:		T_CRYO_PUMP_ATM2303M_STAT;	


	// Input signals
	i_bReady		AT %I*:	BOOL;	// OK for Process, i.e. speed ≥ nominal speed
	i_bSpeed100		AT %I*:	BOOL;	// pump speed > 100 rpm
	i_bWarning		AT %I*:	BOOL;	// presence of a warning
	i_bAlarm		AT %I*:	BOOL;	// presence of an alarm

END_VAR


// Execute the base class object FB_CRYO_PUMP_SERIAL
SUPER^();

METHOD M_Configure
VAR_INPUT
END_VAR
VAR
	//
	// List of INIT commands.
	//
	cmdList_Init_ATH2303M:	ARRAY [1..8] OF T_CRYO_PUMP_CMD := [
		(cmd := cfg.C_CMD_IDN, 	length := 0),	// 29?
		(cmd := cfg.C_CMD_RDI, 	length := 0),	// 11?
		(cmd := cfg.C_CMD_VER, 	length := 92),
		(cmd := '', 		length := 0),
		(cmd := '', 		length := 0),
		(cmd := '', 		length := 0),
		(cmd := '', 		length := 0),
		(cmd := '', 		length := 0)];

	//
	//	List of READ (and WRITE) commands.
	// NOTE: Monitoring loop stops on first cmd = ''.
	//
	cmdList_Read_ATH2303M:	ARRAY [1..16] OF T_CRYO_PUMP_CMD := [
		(cmd := cfg.C_CMD_SEL, 	length := 15),
		(cmd := cfg.C_CMD_STA, 	length := 78),
		(cmd := cfg.C_CMD_LEV, 	length := 66),
		(cmd := '', 		length := 0),
		(cmd := '', 		length := 0),
		(cmd := '', 		length := 0),
		(cmd := '', 		length := 0),
		(cmd := '', 		length := 0),
		(cmd := '', 		length := 0),
		(cmd := '', 		length := 0),
		(cmd := '', 		length := 0),
		(cmd := '', 		length := 0),
		(cmd := '', 		length := 0),
		(cmd := '', 		length := 0),
		(cmd := '', 		length := 0),
		(cmd := '', 		length := 0)];
	
END_VAR
IF NOT bStarted	THEN
	//
	// START: Mandatory for ALL pumps !!!
	//
	// Set references from FB_RS_BASE
	cfgRef	REF=cfg;
	ctrlRef	REF=ctrl;
	statRef	REF=stat;

	// Set references from FB_CRYO_TMP_BASE
	cfgBaseRef	REF=cfg;
	ctrlBaseRef	REF=ctrl;
	statBaseRef	REF=stat;

	// Copy input parameters to configuration
	cfg.nModel			:= in_nModel;
	cfg.bAutoMonitor	:= in_bAutoMonitor;
	cfg.tDelay_Periodic	:= DINT_TO_TIME(in_nPeriod);
	
	
	// Set pointers to arrays of commands
	ptrInitCmds	:= ADR(cfg.cmdList_Init);(* Pointer to INIT commands *)
	ptrReadCmds	:= ADR(cfg.cmdList_Read);(* Pointer to READ commands *)
	
	// TODO in FB that extends the functionality
	// Set pointers to comm, i.e.
	ptrCommCfg	:= ADR(comm.cfg);	(* Pointer to comm.cfg instance *)
	ptrCommCtrl	:= ADR(comm.ctrl);	(* Pointer to comm.ctrl instance *)
	ptrCommStat	:= ADR(comm.stat);	(* Pointer to comm.stat instance *)
	
	// Set comm suffixes for commands and replies
	ptrCommCfg^.sCmdSuffix		:= in_sCmdSuffix;
	ptrCommCfg^.sReplySuffix	:= in_sReplySuffix;

	statRef.bConfigured	:= TRUE;
	bStarted			:= TRUE;
	//
	// END: Mandatory for ALL pumps !!!
	//


	//
	// ATH specific configuration
	//
	
	// Assign INIT and READ commands.
	cfg.cmdList_Init	:= cmdList_Init_ATH2303M;
	cfg.cmdList_Read	:= cmdList_Read_ATH2303M;
END_IF
END_METHOD

METHOD M_GetSpeed : DINT
VAR_INPUT
END_VAR
M_GetSpeed	:= stat.nPumpSpeed;
END_METHOD

METHOD M_IsReady : BOOL
VAR_INPUT
END_VAR
M_IsReady	:= stat.bReady;
END_METHOD

METHOD M_IsRunning : BOOL
VAR_INPUT
END_VAR
M_IsRunning	:= stat.bMoving;
END_METHOD

METHOD M_ReadFromReply : BOOL
// Method to check correctness of the reply and assign the result to a status variable.
VAR_INPUT
	idx:		INT;		(* arr [idx] will hold the first extracted value, arr [idx+1] the second one, etc. *)
	bInitCmd:	BOOL := FALSE;
END_VAR
VAR
	pos:	INT;
	cmd:	STRING;
	length:	DINT;
	subStr:	STRING(255);
END_VAR
// During INIT it might happen that the command index is 0.
// These cases should be discarded.
IF idx <= 0	THEN
	M_ReadFromReply	:= TRUE;
	RETURN;
END_IF

IF bInitCmd	THEN
	cmd		:= cfg.cmdList_Init[idx].cmd;
	length	:= cfg.cmdList_Init[idx].length;
ELSE
	cmd		:= cfg.cmdList_Read[idx].cmd;
	length	:= cfg.cmdList_Read[idx].length;
END_IF

IF length <> 0  AND  LEN(stat.sReply) <> length THEN
	M_ReadFromReply	:= FALSE;
	RETURN;
END_IF

IF cmd = cfg.C_CMD_STA	THEN
	stat.nPumpSpeed		:= STRING_TO_DINT(MID(stat.sReply,5,10));
	stat.nMotorVolt		:= STRING_TO_DINT(MID(stat.sReply,2,36));
	stat.nMotorCurr		:= STRING_TO_DINT(MID(stat.sReply,5,39));
	stat.nPumpTemp		:= STRING_TO_DINT(MID(stat.sReply,3,45));
	stat.nElecTemp	:= STRING_TO_DINT(MID(stat.sReply,3,49));
ELSIF cmd = cfg.C_CMD_LEV	THEN
	stat.nNominalSpeed				:= STRING_TO_DINT(MID(stat.sReply,5,6));
	stat.nStandbySpeed				:= STRING_TO_DINT(MID(stat.sReply,5,12));
	stat.nPumpHours					:= STRING_TO_DINT(MID(stat.sReply,5,26));
	stat.nElecHours					:= STRING_TO_DINT(MID(stat.sReply,5,32));
	stat.nSetPoint_AtSpeed			:= STRING_TO_DINT(MID(stat.sReply,2,54));
	stat.nSetPoint_Temp				:= STRING_TO_DINT(MID(stat.sReply,2,57));
	stat.nSetPoint_BearingWarn		:= STRING_TO_DINT(MID(stat.sReply,2,60));
	stat.nSetPoint_BearingCounter	:= STRING_TO_DINT(MID(stat.sReply,3,63));
ELSIF cmd = cfg.C_CMD_IDN	THEN
	stat.sIDN	:= MID(stat.sReply, LEN(stat.sReply)-6, 6);	// Strip the string off prefix and sufix.
ELSIF cmd = cfg.C_CMD_RDI	THEN
	stat.sRDI	:= MID(stat.sReply, LEN(stat.sReply)-6, 6);	// Strip the string off prefix and sufix.
ELSIF cmd = cfg.C_CMD_VER	THEN
	subStr		:= MID(stat.sReply, LEN(stat.sReply)-6, 6);	// Strip the string off prefix and sufix.
	pos			:= FIND(subStr, ',');	// Find first comma
	stat.sVer1	:= MID(subStr, pos-1, 1);	// Assign substring up to the first comma char
	subStr		:= MID(subStr, LEN(subStr)-pos, pos+1);	// Take the string after sVer1 and comma.
	pos			:= FIND(subStr, ',');	// Find next comma
	stat.sVer2	:= MID(subStr, pos-1, 1);	// Take the string up to the comma
	subStr		:= MID(subStr, LEN(subStr)-pos, pos+1);	// Take the string after sVer1 and comma.
	pos			:= FIND(subStr, ',');	// Find next comma
	stat.sVer3	:= MID(subStr, pos-1, 1);	// Take the string up to the comma
	subStr		:= MID(subStr, LEN(subStr)-pos, pos+1);	// Take the string after sVer1 and comma.
	stat.sVer4	:= subStr;	// Take the rest as sVer4
ELSIF cmd = cfg.C_CMD_SEL	THEN
	stat.nCtrlMode		:= STRING_TO_DINT(MID(stat.sReply,1,14));
END_IF


M_ReadFromReply	:= true;	// OK
END_METHOD

METHOD M_UpdateStatus
VAR_INPUT
END_VAR
// Update Status from digital inputs readings
stat.bReady		:= i_bReady;
stat.bSpeed100	:= i_bSpeed100;
stat.bWarning	:= NOT i_bWarning;	// Active low
stat.bAlarm		:= NOT i_bAlarm;	// Active low

stat.bMoving	:= stat.bReady OR stat.bSpeed100 OR stat.nPumpSpeed > 0;

// Set Control Mode Label
CASE stat.nCtrlMode	OF
	0:	stat.sCtrlMode	:= 'HHR (Hand-Held Remote)';
	1:	stat.sCtrlMode	:= 'REMOTE';
	2:	stat.sCtrlMode	:= 'SERIAL LINK';
	3:	stat.sCtrlMode	:= 'FIELDBUS';
ELSE
	stat.sCtrlMode	:= 'UNKNOWN';
END_CASE
END_METHOD

END_FUNCTION_BLOCK

// ---- POUs/Subsystems/Examples/Evacuation/FB_CRYO_EVAC_MICADO.TcPOU
FUNCTION_BLOCK FB_CRYO_EVAC_MICADO EXTENDS FB_CRYO_EVAC_BASE_50000
VAR_INPUT
END_VAR
VAR_OUTPUT
END_VAR
VAR
	// Specify pumps
	rp:	FB_CRYO_PUMP_ECODRY;	// Roughing Pump
	tp:	FB_CRYO_PUMP_ATH2303M;	// Turbomolecular Pump
	
END_VAR

SUPER^();	// Execute base FB code.

METHOD M_Configure
VAR_INPUT
END_VAR
//
// Specific MICADO configuration.
//
IF NOT stat.bConfigured	THEN
	//
	// MANDATORY !!!
	// Call base FB::M_Configure() to set the pointers.
	//
	SUPER^.M_Configure();
	

	// MANDATORY: Set References for pumps!!!
	// If not done, system will crash !!!
	rpRef	REF=rp;
	tpRef	REF=tp;
	

	// Specific instance configuration, e.g. anything different
	// from the default values given in the cfg structure of type T_CRYO_EVAC_CFG_50000.
	cfg.nType_VAG1	:= E_CRYO_SENSOR_TYPE_PRESS.WRG_D_NW25;
	cfg.nType_VAG2	:= E_CRYO_SENSOR_TYPE_PRESS.WRG_D_NW25;
	cfg.nType_VAG3	:= E_CRYO_SENSOR_TYPE_PRESS.WRG_D_NW25;
	cfg.nType_VAGF1	:= E_CRYO_SENSOR_TYPE_PRESS.PKR_250;
	cfg.nType_VAGF2	:= E_CRYO_SENSOR_TYPE_PRESS.PKR_250;
	cfg.nType_VAGG1	:= E_CRYO_SENSOR_TYPE_PRESS.PKR_250;
	cfg.nType_VAGG2	:= E_CRYO_SENSOR_TYPE_PRESS.PKR_250;


	stat.bConfigured	:= TRUE;
ELSE
	RETURN;	// Nothing to do any more
END_IF
END_METHOD

METHOD M_ExecuteControllers
VAR_INPUT
END_VAR
//
// Specific MICADO Evacuation System HW configuration.
//

// Roughing Pump	
rp(	
	in_bSimulation	:= FALSE,
	in_sName		:= 'ECODRY V01',
	in_bEnable		:= ctrl.bEnable_PVP,
	in_nSlaveID		:= 31,
	in_sVersion		:= 'V01',
	in_nPeriod		:= 2000);

// Turbo Molecular Pump
tp(	
	in_bSimulation	:= FALSE,
	in_sName		:= 'ATH2303M',
	in_bEnable		:= ctrl.bEnable_TMP,
	in_nModel		:= 2303,
	in_bAutoMonitor	:= TRUE,
	in_nPeriod		:= 2000);

// Valves are controlled in the base FB
SUPER^.M_ExecuteControllers();
END_METHOD

END_FUNCTION_BLOCK

// ---- POUs/Subsystems/Evacuation/FB_CRYO_EVAC_BASE_50000.TcPOU
FUNCTION_BLOCK FB_CRYO_EVAC_BASE_50000
VAR_INPUT
	in_bEnable:		BOOL := FALSE;	// System active while in_bEnable is TRUE
	in_RefVAGF:		REFERENCE TO FB_CRYO_PRESSURE_VOTE;
	in_RefVAGG:		REFERENCE TO FB_CRYO_PRESSURE_VOTE;
END_VAR
VAR_OUTPUT
END_VAR
VAR
	/////////
	// Pumps
	/////////
	
	rpRef:	REFERENCE TO FB_CRYO_PUMP_BASE;		// Roughing Pump
	tpRef:	REFERENCE TO FB_CRYO_PUMP_BASE;		// Turbo Molecular Pump
	
	//////////
	// Valves
	//////////
	
	PVV1:	FB_CRYO_VALVE_CTRL;					// Prevacuum Valve #1
	PVV2:	FB_CRYO_VALVE_CTRL;					// Prevacuum Valve #2
	PVV3:	FB_CRYO_VALVE_CTRL;					// Prevacuum Valve #3
	PVV4:	FB_CRYO_VALVE_CTRL;					// Prevacuum Valve #4
	GBV:	FB_CRYO_VALVE_CTRL;					// Gas-ballast Valve
	
	// Valve command handling
	cmdPVV1:	FB_CRYO_ACTUATOR_CMD;
	cmdPVV2:	FB_CRYO_ACTUATOR_CMD;
	cmdPVV3:	FB_CRYO_ACTUATOR_CMD;
	cmdPVV4:	FB_CRYO_ACTUATOR_CMD;
	cmdGBV:		FB_CRYO_ACTUATOR_CMD;

	
	// Pointers to valves
	ptrV:	ARRAY [1..5] OF POINTER TO FB_CRYO_VALVE_CTRL;
	// Pointers to valve commands
	ptrVC:	ARRAY [1..5] OF POINTER TO FB_CRYO_ACTUATOR_CMD;
	// Pointers to Enable flags for valves
	ptrEV:	ARRAY [1..5] OF POINTER TO BOOL;
	
	////////////
	// Pressure
	////////////
	
	// Pressure transducers
	sensor_VAG1:	FB_CRYO_SENSOR_PRESSURE;	// Prevacuum pressure gauge #1
	sensor_VAG2:	FB_CRYO_SENSOR_PRESSURE;	// Prevacuum pressure gauge #2
	sensor_VAG3:	FB_CRYO_SENSOR_PRESSURE;	// Prevacuum pressure gauge #3

	
	// Pressure measurements
	VAG1:	FB_CRYO_PRESSURE_VOTE;				// Prevacuum pressure #1
	VAG2:	FB_CRYO_PRESSURE_VOTE;				// Prevacuum pressure #2
	VAG3:	FB_CRYO_PRESSURE_VOTE;				// Prevacuum pressure #3
	VAGF:	FB_CRYO_PRESSURE_VOTE;				// Cryo pressure F
	VAGG:	FB_CRYO_PRESSURE_VOTE;				// Cryo pressure G
	// Pointers to pressures
	ptrP:	ARRAY [1..5] OF POINTER TO FB_CRYO_PRESSURE_VOTE;
	
	
	cfg:	T_CRYO_EVAC_CFG_50000;
	ctrl:	T_CRYO_EVAC_CTRL_50000;
	stat:	T_CRYO_EVAC_STAT_50000;
	
	timer:	TON;
	trig:	R_TRIG;	// Start trigger
	
	// GUI staff
	guiValveIndex:	UINT := 1;	// Index for Valve Engineering GUI
END_VAR

// NOTE: Configuration is set on the first cycle.
//       Once stat.bConfigured is TRUE, 
//       configuration is not updated any more.
M_Configure();

M_ReadSensors();

M_ExecuteControllers();

M_UpdateStatus();

M_StateMachine();

METHOD M_ActionExecute
VAR_INPUT
END_VAR
CASE stat.nState	OF
	E_CRYO_EVAC_STATE_50000.NONE:
		;	// Nothing to do

	E_CRYO_EVAC_STATE_50000.OFF:
		;	// Nothing to do

	E_CRYO_EVAC_STATE_50000.START_PVP:
		ctrl.bEnable_PVP	:= TRUE;
		ctrl.bEnable_PVV1	:= FALSE;
		ctrl.bEnable_PVV2	:= FALSE;
		ctrl.bEnable_PVV3	:= FALSE;
		ctrl.bEnable_PVV4	:= FALSE;
		ctrl.bEnable_GBV	:= FALSE;

	E_CRYO_EVAC_STATE_50000.OPEN_GBV:
		ctrl.bEnable_GBV	:= TRUE;

	E_CRYO_EVAC_STATE_50000.WAIT_VAG3:
		;	// Nothing to do

	E_CRYO_EVAC_STATE_50000.OPEN_PVV1:
		ctrl.bEnable_PVV1	:= TRUE;

	E_CRYO_EVAC_STATE_50000.WAIT_VAG_1_3:
		;	// Nothing to do

	E_CRYO_EVAC_STATE_50000.OPEN_PVV2:
		ctrl.bEnable_PVV2	:= TRUE;

	E_CRYO_EVAC_STATE_50000.WAIT_VAG_F_G_1:
		;	// Nothing to do

	E_CRYO_EVAC_STATE_50000.CLOSE_PVV2:
		ctrl.bEnable_PVV2	:= FALSE;

	E_CRYO_EVAC_STATE_50000.CLOSE_PVV1:
		ctrl.bEnable_PVV1	:= FALSE;

	E_CRYO_EVAC_STATE_50000.START_TMP:
		ctrl.bEnable_TMP	:= TRUE;
		
	E_CRYO_EVAC_STATE_50000.OPEN_PVV3:
		ctrl.bEnable_PVV3	:= TRUE;

	E_CRYO_EVAC_STATE_50000.WAIT_VAG_2_3:
		;	// Nothing to do

	E_CRYO_EVAC_STATE_50000.OPEN_PVV4:
		ctrl.bEnable_PVV4	:= TRUE;

	E_CRYO_EVAC_STATE_50000.WAIT_VAG_F_G_2:
		;	// Nothing to do

	E_CRYO_EVAC_STATE_50000.CLOSE_GBV:
		ctrl.bEnable_GBV	:= FALSE;

	E_CRYO_EVAC_STATE_50000.EVACUATING:
		;	// Nothing to do

	E_CRYO_EVAC_STATE_50000.CLOSE_ALL_VALVES:
		ctrl.bEnable_PVV1	:= FALSE;
		ctrl.bEnable_PVV2	:= FALSE;
		ctrl.bEnable_PVV3	:= FALSE;
		ctrl.bEnable_PVV4	:= FALSE;
		ctrl.bEnable_GBV	:= FALSE;

	E_CRYO_EVAC_STATE_50000.DELAY_STOPPING:
		;	// Nothing to do

	E_CRYO_EVAC_STATE_50000.STOP_TMP_1:
		ctrl.bEnable_TMP	:= FALSE;

	E_CRYO_EVAC_STATE_50000.STOP_PVP:
		ctrl.bEnable_PVP	:= FALSE;

	E_CRYO_EVAC_STATE_50000.WAIT_TMP_STANDSTILL:
		;	// Nothing to do

	E_CRYO_EVAC_STATE_50000.STOP_TMP_2:
		ctrl.bEnable_TMP	:= FALSE;
	
END_CASE

timer(IN:=FALSE);	// Reset timer, just in case.
END_METHOD

METHOD M_Activity_ClosingAllValves
VAR_INPUT
END_VAR
VAR
	i:			INT;
	bAllClosed:	BOOL := TRUE;
END_VAR
// Check all valves if they are closed.
// If any of them is not closed, then they are not all closed.
FOR i := 1 TO 5 DO
	IF NOT ptrV[i]^.stat.bActOFF	THEN
		bAllClosed	:= FALSE;
		EXIT;
	END_IF
END_FOR

IF bAllClosed THEN
	// All valves are closed.
	// In next state apply a delay before stopping pumps.
	M_SetNextState(E_CRYO_EVAC_STATE_50000.DELAY_STOPPING);
END_IF
END_METHOD

METHOD M_Activity_ClosingValve
VAR_INPUT
	index:		INT;
	nNextState:	E_CRYO_EVAC_STATE_50000;	// Next state after valve is closed
END_VAR
// Check if valve index is valid.
// If not, just return (for safety).
IF index < 1  OR  index > 5	THEN
	RETURN;
END_IF 

IF ptrV[index]^.stat.bActOFF THEN
	// The valve is closed.
	// Set next state and execute its action
	M_SetNextState(nNextState);	// Next state
	
END_IF
END_METHOD

METHOD M_Activity_DelayBeforeStoppingPumps
VAR_INPUT
END_VAR
timer(IN:=TRUE, PT:=CFG.tDelay);

IF timer.Q THEN
	// Delay timer expired.
	// Reset timer.
	timer(IN:=FALSE);
	
	// Stop Turbo Pump.
	M_SetNextState(E_CRYO_EVAC_STATE_50000.STOP_TMP_1);	// Next state

END_IF
END_METHOD

METHOD M_Activity_Evacuating
VAR_INPUT
END_VAR
VAR
	index1:	INT	:= E_CRYO_EVAC_PRESSURES_50000.VAG2;
	index2:	INT	:= E_CRYO_EVAC_PRESSURES_50000.VAG3;
END_VAR
// System is started by setting in_bEnable to TRUE
IF NOT in_bEnable THEN
	// If system is disabled, start stopping procedure.
	M_SetNextState(E_CRYO_EVAC_STATE_50000.CLOSE_ALL_VALVES);	// Next state
	
ELSIF 	ptrP[index1]^.stat.lrPressure > cfg.lrThld_PrevacHigh  AND
		ptrP[index2]^.stat.lrPressure > cfg.lrThld_PrevacHigh THEN
	// Something is wrong. Prevacuum pressure is too high. Stop evacuation!
	// Set error.
	M_SetError('Prevacuum pressure too high. Stopping evacuation...');
	M_SetNextState(E_CRYO_EVAC_STATE_50000.CLOSE_ALL_VALVES);	// Next state
	
END_IF
END_METHOD

METHOD M_Activity_Off
VAR_INPUT
END_VAR
// Disable anything that is not safe in this state
ctrl.bEnable_PVP	:= FALSE;
ctrl.bEnable_TMP	:= FALSE;
ctrl.bEnable_PVV1	:= FALSE;
ctrl.bEnable_PVV2	:= FALSE;
ctrl.bEnable_PVV3	:= FALSE;
ctrl.bEnable_PVV4	:= FALSE;
ctrl.bEnable_GBV	:= FALSE;


// System is started by setting in_bEnable to TRUE
trig(CLK := in_bEnable);

IF trig.Q THEN
	// Clear any existing error
	M_SetError('OK');
	
	M_SetNextState(E_CRYO_EVAC_STATE_50000.START_PVP);	// Next state
END_IF
END_METHOD

METHOD M_Activity_OpeningValve
VAR_INPUT
	index:		INT;
	nNextState:	E_CRYO_EVAC_STATE_50000;	// Next state after valve is closed
END_VAR
IF NOT in_bEnable THEN
	// If system is disabled, start stopping procedure.
	M_SetNextState(E_CRYO_EVAC_STATE_50000.CLOSE_ALL_VALVES);	// Next state
	
ELSIF ptrV[index]^.stat.bActON THEN
	// The valve is open.
	// Go to next state
	M_SetNextState(nNextState);
	
END_IF
END_METHOD

METHOD M_Activity_StartingPVP
VAR_INPUT
END_VAR
// Disable anything that is not safe in this state
ctrl.bEnable_TMP	:= FALSE;
ctrl.bEnable_PVV1	:= FALSE;
ctrl.bEnable_PVV2	:= FALSE;
ctrl.bEnable_PVV3	:= FALSE;
ctrl.bEnable_PVV4	:= FALSE;
ctrl.bEnable_GBV	:= FALSE;


IF NOT in_bEnable THEN
	// If system is disabled, start stopping procedure.
	M_SetNextState(E_CRYO_EVAC_STATE_50000.CLOSE_ALL_VALVES);	// Next state
	
ELSIF rpRef.M_IsReady() THEN
	// Roughing Pump is Ready.
	// Open Gas-ballast valve.
	M_SetNextState(E_CRYO_EVAC_STATE_50000.OPEN_GBV);	// Next state
	
END_IF
END_METHOD

METHOD M_Activity_StartingTMP
VAR_INPUT
END_VAR
VAR
	index1:	INT	:= E_CRYO_EVAC_PRESSURES_50000.VAGF;
	index2:	INT	:= E_CRYO_EVAC_PRESSURES_50000.VAGG;
END_VAR
IF NOT in_bEnable THEN
	// If system is disabled, start stopping procedure by closing all valves.
	M_SetNextState(E_CRYO_EVAC_STATE_50000.CLOSE_ALL_VALVES);	// Next state
	
ELSIF 	ptrP[index1]^.stat.lrPressure > cfg.lrThld_Prevac  OR
		ptrP[index2]^.stat.lrPressure > cfg.lrThld_Prevac 	THEN
	// Cryostat pressure is too high for some reason.
	// Stop Turbo Molecular pump.
	M_SetNextState(E_CRYO_EVAC_STATE_50000.STOP_TMP_2);
		
ELSIF tpRef.M_IsReady() THEN
	// Turbo Molecular Pump is Ready, i.e., running at operational speed.
	// Open PVV3.
	M_SetNextState(E_CRYO_EVAC_STATE_50000.OPEN_PVV3);	// Next state
	
END_IF
END_METHOD

METHOD M_Activity_StoppingPVP
VAR_INPUT
END_VAR
// Disable anything that is not safe in this state
ctrl.bEnable_PVP	:= FALSE;
ctrl.bEnable_TMP	:= FALSE;


// The evacuation system is in the process of shutting down.
// Allow re-starting of evacuation.
// System is started by setting in_bEnable to TRUE.
trig(CLK := in_bEnable);

IF trig.Q THEN
	// Clear any existing error
	M_SetError('OK');
	
	// Enable Roughing Pump
	M_SetNextState(E_CRYO_EVAC_STATE_50000.START_PVP);
	
ELSIF NOT rpRef.M_IsRunning() THEN
	// The Roughing Pump stopped.
	// Wait for the Turbo Pump to get to complete stop.
	M_SetNextState(E_CRYO_EVAC_STATE_50000.WAIT_TMP_STANDSTILL);	// Next state

END_IF
END_METHOD

METHOD M_Activity_StoppingTMP
VAR_INPUT
	index:	INT;	// Index of action(1 or 2, for STP_TMP and STOP2_TMP)
END_VAR
// Disable anything that is not safe in this state


// The evacuation system is in the process of shutting down.
// Allow re-starting of evacuation.
// System is started by setting in_bEnable to TRUE.
trig(CLK := in_bEnable);

IF trig.Q THEN
	// Clear any existing error
	M_SetError('OK');
	
	// Enable Roughing Pump
	M_SetNextState(E_CRYO_EVAC_STATE_50000.START_PVP);
	
ELSIF NOT tpRef.M_IsReady() THEN
	// TODO: This is ATH2303M specific.
	//       Maybe, speed < 100 or similar check.
	
	IF index = 1	THEN
		// Case 1: Proceed with stopping PVP.
		M_SetNextState(E_CRYO_EVAC_STATE_50000.STOP_PVP);
	ELSIF index = 2	THEN
		// Case 2: Proceed with openning PVV1.
		M_SetNextState(E_CRYO_EVAC_STATE_50000.OPEN_PVV1);
	END_IF
	
END_IF
END_METHOD

METHOD M_Activity_Waiting2Pressures
VAR_INPUT
	index1:		INT;
	index2:		INT;
	lrRef:		LREAL;	// Reference pressure [mbar]
	nNextState:	E_CRYO_EVAC_STATE_50000;	// Next state after pressure is reached
END_VAR
// Check if valve indexes are valid. Range [1..5]
// If not, just return (for safety).
IF index1 < 1  OR  index1 > 5  OR  index2 < 1  OR  index2 > 5  THEN
	RETURN;
END_IF 

IF	(ptrP[index1]^.stat.bValid  AND  ptrP[index1]^.stat.lrPressure < lrRef)  AND
	(ptrP[index2]^.stat.bValid  AND  ptrP[index2]^.stat.lrPressure < lrRef)  	THEN
	// The pressure has been reached.
	
	M_SetNextState(nNextState);	// Next state
END_IF
END_METHOD

METHOD M_Activity_WaitingPressure
VAR_INPUT
	index:		INT;
	lrRef:		LREAL;	// Reference pressure [mbar]
	nNextState:	E_CRYO_EVAC_STATE_50000;	// Next state after pressure is reached
END_VAR
// Check if valve index is valid.
// If not, just return (for safety).
IF index < 1  OR  index > 5	THEN
	RETURN;
END_IF 

IF ptrP[index]^.stat.bValid  AND  ptrP[index]^.stat.lrPressure < lrRef  THEN
	// The pressure has been reached.
	
	M_SetNextState(nNextState);	// Next state
END_IF
END_METHOD

METHOD M_Activity_WaitingTMP2Stop
VAR_INPUT
END_VAR
// Disable anything that is not safe in this state
ctrl.bEnable_PVP	:= FALSE;
ctrl.bEnable_TMP	:= FALSE;


// The evacuation system is in the process of shutting down.
// Allow re-starting of evacuation.
// System is started by setting in_bEnable to TRUE.
trig(CLK := in_bEnable);

IF trig.Q THEN
	// Clear any existing error
	M_SetError('OK');
	
	// Enable Roughing Pump
	M_SetNextState(E_CRYO_EVAC_STATE_50000.START_PVP);
	
ELSIF tpRef.M_GetSpeed() = 0 THEN
	// The Turbo Pump came to complete stop.
	// The Evacuation system is OFF.
	M_SetNextState(E_CRYO_EVAC_STATE_50000.OFF);
	
END_IF
END_METHOD

METHOD M_Configure
VAR_INPUT
END_VAR
//
// TODO USER: 
// This M_Configure() MUST be called once in the child FB M_Configure() method!!!
// It sets all the pointers to various variables.
// 
(*
//
// TODO USER in child FB
//
	// MANDATORY: Set References to pumps!!!
	// If not done, system will crash !!!
	rpRef	REF=rp;
	tpRef	REF=tp;
	
	// Specific instance configuration, e.g. pressure gauges' types.
	// See FB_CRYO_EVAC_MICADO::M_Configure().
	// ...

*)	

// Set pointers to Valves - MUST!!!
ptrV[1]	:= ADR(PVV1);
ptrV[2]	:= ADR(PVV2);
ptrV[3]	:= ADR(PVV3);
ptrV[4]	:= ADR(PVV4);
ptrV[5]	:= ADR(GBV);

// Set pointers to Valve Commands - MUST!!!
ptrVC[1]	:= ADR(cmdPVV1);
ptrVC[2]	:= ADR(cmdPVV2);
ptrVC[3]	:= ADR(cmdPVV3);
ptrVC[4]	:= ADR(cmdPVV4);
ptrVC[5]	:= ADR(cmdGBV);

// Set pointers to Enable Valves flags - MUST!!!
ptrEV[1]	:= ADR(ctrl.bEnable_PVV1);
ptrEV[2]	:= ADR(ctrl.bEnable_PVV2);
ptrEV[3]	:= ADR(ctrl.bEnable_PVV3);
ptrEV[4]	:= ADR(ctrl.bEnable_PVV4);
ptrEV[5]	:= ADR(ctrl.bEnable_GBV);


// Set pointers to Pressures - MUST!!!
ptrP[1]	:= ADR(VAG1);
ptrP[2]	:= ADR(VAG2);
ptrP[3]	:= ADR(VAG3);
ptrP[4]	:= ADR(VAGF);
ptrP[5]	:= ADR(VAGG);
END_METHOD

METHOD M_ExecuteControllers
VAR_INPUT
END_VAR
// Valve commands
cmdPVV1(in_bEnable := ctrl.bEnable_PVV1);	// Handling of PVV1 commands
cmdPVV2(in_bEnable := ctrl.bEnable_PVV2);	// Handling of PVV2 commands
cmdPVV3(in_bEnable := ctrl.bEnable_PVV3);	// Handling of PVV3 commands
cmdPVV4(in_bEnable := ctrl.bEnable_PVV4);	// Handling of PVV4 commands
cmdGBV (in_bEnable := ctrl.bEnable_GBV);	// Handling of GBV  commands

// Valve Control
PVV1(
	in_bEnable			:= cmdPVV1.out_bEnable,
	in_nFeedback		:= E_CRYO_BIN_ACT_FEEDBACK.ON_AND_OFF);

PVV2(
	in_bEnable			:= cmdPVV2.out_bEnable,
	in_nFeedback		:= E_CRYO_BIN_ACT_FEEDBACK.ON_AND_OFF);

PVV3(
	in_bEnable			:= cmdPVV3.out_bEnable,
	in_nFeedback		:= E_CRYO_BIN_ACT_FEEDBACK.ON_AND_OFF);

PVV4(
	in_bEnable			:= cmdPVV4.out_bEnable,
	in_nFeedback		:= E_CRYO_BIN_ACT_FEEDBACK.ON_AND_OFF);

GBV(
	in_bEnable			:= cmdGBV.out_bEnable,
	in_nFeedback		:= E_CRYO_BIN_ACT_FEEDBACK.ON_AND_OFF);
END_METHOD

METHOD M_ReadSensors
VAR_INPUT
END_VAR
///////////////////////////////////////////////
// Read individual prevacuum pressure sensors.
///////////////////////////////////////////////
//
// Pressure readings are averaged over 100 ms.
//
// Note: Pressure sensor type is configured in cfg and overwritten in M_Configure().
//       Default is Pfeiffer PKR 360 KF25.
sensor_VAG1	(in_nType := cfg.nType_VAG1,	in_nSampleTime := 100);
sensor_VAG2	(in_nType := cfg.nType_VAG2,	in_nSampleTime := 100);
sensor_VAG3	(in_nType := cfg.nType_VAG3,	in_nSampleTime := 100);
(*
sensor_VAGF1(in_nType := cfg.nType_VAGF1,	in_nSampleTime := 100);
sensor_VAGF2(in_nType := cfg.nType_VAGF2,	in_nSampleTime := 100);
sensor_VAGG1(in_nType := cfg.nType_VAGG1,	in_nSampleTime := 100);
sensor_VAGG2(in_nType := cfg.nType_VAGG2,	in_nSampleTime := 100);
*)

//////////////////////////////////////////////
// Use voting system to calculate pressures.
//////////////////////////////////////////////
//
// Note: VAG 1-3 have got only one sensor pressure connected !!!
//       VAG F & G have got two pressure sensors connected !
//
VAG1(
	in_bSimulation	:= cfg.bPressSimulation,
	in_nNumSensor	:= 2,
	in_nVoteMethod	:= E_CRYO_VOTE.V_1oo2,
	in_pSensor1		:= ADR(sensor_VAG1));

VAG2(
	in_bSimulation	:= cfg.bPressSimulation,
	in_nNumSensor	:= 2,
	in_nVoteMethod	:= E_CRYO_VOTE.V_1oo2,
	in_pSensor1		:= ADR(sensor_VAG2));

VAG3(
	in_bSimulation	:= cfg.bPressSimulation,
	in_nNumSensor	:= 2,
	in_nVoteMethod	:= E_CRYO_VOTE.V_1oo2,
	in_pSensor1		:= ADR(sensor_VAG3));

	
// Copy pressure references to local variables
VAGF	:= in_RefVAGF;
VAGG	:= in_RefVAGG;

	
(*	
VAGF(
	in_bSimulation	:= cfg.bPressSimulation,
	in_nNumSensor	:= 2,
	in_nVoteMethod	:= E_CRYO_VOTE.V_1oo2,
	in_pSensor1		:= ADR(sensor_VAGF1),
	in_pSensor2		:= ADR(sensor_VAGF2));

VAGG(
	in_bSimulation	:= cfg.bPressSimulation,
	in_nNumSensor	:= 2,
	in_nVoteMethod	:= E_CRYO_VOTE.V_1oo2,
	in_pSensor1		:= ADR(sensor_VAGG1),
	in_pSensor2		:= ADR(sensor_VAGG2));
*)
END_METHOD

METHOD M_SetError
VAR_INPUT
	in_sErrorText:	STRING(64);
END_VAR
stat.bError		:= (in_sErrorText <> 'OK');
stat.sErrorText	:= in_sErrorText;
END_METHOD

METHOD M_SetLabels
VAR_INPUT
END_VAR
VAR
    fbFormat:	FB_FormatString;
	nVal:		UDINT;
	lrVal:		LREAL;
END_VAR
CASE stat.nState	OF
	E_CRYO_EVAC_STATE_50000.NONE:
		stat.sState		:= 'NONE';
		stat.sStatus	:= 'UNKNOWN';
		
	E_CRYO_EVAC_STATE_50000.OFF:
		stat.sState		:= 'OFF';
		stat.sStatus	:= 'OFF';
		
	E_CRYO_EVAC_STATE_50000.START_PVP:
		stat.sState		:= 'START_PVP';
		stat.sStatus	:= 'Starting Roughing Pump...';
		
	E_CRYO_EVAC_STATE_50000.START_TMP:
		stat.sState		:= 'START_TMP';
		stat.sStatus	:= 'Starting Turbo Molecular Pump...';
		
	E_CRYO_EVAC_STATE_50000.STOP_TMP_1,
	E_CRYO_EVAC_STATE_50000.STOP_TMP_2:
		stat.sState		:= 'STOP_TMP_x';
		stat.sStatus	:= 'Stopping Turbo Molecular Pump...';
		
	E_CRYO_EVAC_STATE_50000.STOP_PVP:
		stat.sState		:= 'STOP_PVP';
		stat.sStatus	:= 'Stopping Roughing Pump...';
		
	E_CRYO_EVAC_STATE_50000.WAIT_VAG3:
		stat.sState		:= 'WAIT_VAG3';
		fbFormat(	sFormat := 'Waiting VAG3 <= %.4f [mbar]...', 
					arg1 := F_LREAL(cfg.lrThld_Prevac), 
					sOut => stat.sStatus);
					
	E_CRYO_EVAC_STATE_50000.WAIT_VAG_1_3:
		stat.sState		:= 'WAIT_VAG_1_3';
		fbFormat(	sFormat := 'Waiting VAG1 & VAG3 <= %.4f [mbar]...', 
					arg1 := F_LREAL(cfg.lrThld_Prevac), 
					sOut => stat.sStatus);
					
	E_CRYO_EVAC_STATE_50000.WAIT_VAG_2_3:
		stat.sState		:= 'WAIT_VAG_2_3';
		fbFormat(	sFormat := 'Waiting VAG2 & VAG3 <= %.4f [mbar]...', 
					arg1 := F_LREAL(cfg.lrThld_Prevac), 
					sOut => stat.sStatus);
					
	E_CRYO_EVAC_STATE_50000.WAIT_VAG_F_G_1:
		stat.sState		:= 'WAIT_VAG_F_G_1';
		lrVal			:= 0.9 * cfg.lrThld_Prevac;
		fbFormat(	sFormat := 'Waiting VAGF & VAGG <= %.4f [mbar]...', 
					arg1 := F_LREAL(lrVal), 
					sOut => stat.sStatus);
					
	E_CRYO_EVAC_STATE_50000.WAIT_VAG_F_G_2:
		stat.sState		:= 'WAIT_VAG_F_G_2';
		fbFormat(	sFormat := 'Waiting VAGF & VAGG <= %.4f [mbar]...', 
					arg1 := F_LREAL(cfg.lrThld_Vacuum), 
					sOut => stat.sStatus);
					
	E_CRYO_EVAC_STATE_50000.OPEN_PVV1:
		stat.sState		:= 'OPEN_PVV1';
		stat.sStatus	:= 'Opening PVV1 Valve...';

	E_CRYO_EVAC_STATE_50000.OPEN_PVV2:
		stat.sState		:= 'OPEN_PVV2';
		stat.sStatus	:= 'Opening PVV2 Valve...';

	E_CRYO_EVAC_STATE_50000.OPEN_PVV3:
		stat.sState		:= 'OPEN_PVV3';
		stat.sStatus	:= 'Opening PVV3 Valve...';

	E_CRYO_EVAC_STATE_50000.OPEN_PVV4:
		stat.sState		:= 'OPEN_PVV4';
		stat.sStatus	:= 'Opening PVV4 Valve...';
	
	E_CRYO_EVAC_STATE_50000.OPEN_GBV:
		stat.sState		:= 'OPEN_GBV';
		stat.sStatus	:= 'Opening Gas-ballast Valve...';

	E_CRYO_EVAC_STATE_50000.CLOSE_PVV1:
		stat.sState		:= 'CLOSE_PVV1';
		stat.sStatus	:= 'Closing PVV1 Valve...';

	E_CRYO_EVAC_STATE_50000.CLOSE_PVV2:
		stat.sState		:= 'CLOSE_PVV2';
		stat.sStatus	:= 'Closing PVV2 Valve...';

	E_CRYO_EVAC_STATE_50000.CLOSE_GBV:
		stat.sState		:= 'CLOSE_GBV';
		stat.sStatus	:= 'Closing GBV Valve...';

	E_CRYO_EVAC_STATE_50000.CLOSE_ALL_VALVES:
		stat.sState		:= 'CLOSE_ALL_VALVES';
		stat.sStatus	:= 'Closing All Valves...';
		
	E_CRYO_EVAC_STATE_50000.EVACUATING:
		stat.sState		:= 'EVACUATING';
		stat.sStatus	:= 'EVACUATING...';
		
	E_CRYO_EVAC_STATE_50000.DELAY_STOPPING:
		stat.sState		:= 'DELAY_STOPPING';
		nVal			:= TIME_TO_UDINT(cfg.tDelay);
		fbFormat(	sFormat := 'Delay of %d [ms] Before Stopping Pumps...', 
					arg1 := F_UDINT(nVal), 
					sOut => stat.sStatus);
					
	E_CRYO_EVAC_STATE_50000.WAIT_TMP_STANDSTILL:
		stat.sState		:= 'WAIT_TMP_STANDSTILL';
		stat.sStatus	:= 'Waiting for Turbo Molecular Pump to get Standstill...';
	
END_CASE
END_METHOD

METHOD M_SetNextState
VAR_INPUT
	nNextState:	E_CRYO_EVAC_STATE_50000;	// Next state
END_VAR
stat.nState	:= nNextState;	// Next state
M_ActionExecute();			// Execute Action for next state
M_SetLabels();
END_METHOD

METHOD M_StateMachine
VAR_INPUT
END_VAR
CASE stat.nState	OF
	E_CRYO_EVAC_STATE_50000.NONE:
		M_SetNextState(E_CRYO_EVAC_STATE_50000.OFF);
	E_CRYO_EVAC_STATE_50000.OFF:
		M_Activity_Off();

	E_CRYO_EVAC_STATE_50000.START_PVP:
		M_Activity_StartingPVP();

	E_CRYO_EVAC_STATE_50000.OPEN_GBV:
		M_Activity_OpeningValve(
			index		:= E_CRYO_EVAC_VALVES_50000.GBV, 
			nNextState	:= E_CRYO_EVAC_STATE_50000.WAIT_VAG3);

	E_CRYO_EVAC_STATE_50000.WAIT_VAG3:
		M_Activity_WaitingPressure(
			index		:= E_CRYO_EVAC_PRESSURES_50000.VAG3, 
			lrRef		:= cfg.lrThld_Prevac, 
			nNextState	:= E_CRYO_EVAC_STATE_50000.OPEN_PVV1);

	E_CRYO_EVAC_STATE_50000.OPEN_PVV1:
		M_Activity_OpeningValve(
			index		:= E_CRYO_EVAC_VALVES_50000.PVV1, 
			nNextState	:= E_CRYO_EVAC_STATE_50000.WAIT_VAG_1_3);

	E_CRYO_EVAC_STATE_50000.WAIT_VAG_1_3:
		M_Activity_Waiting2Pressures(
			index1		:= E_CRYO_EVAC_PRESSURES_50000.VAG1, 
			index2		:= E_CRYO_EVAC_PRESSURES_50000.VAG3, 
			lrRef		:= cfg.lrThld_Prevac, 
			nNextState	:= E_CRYO_EVAC_STATE_50000.OPEN_PVV2);

	E_CRYO_EVAC_STATE_50000.OPEN_PVV2:
		M_Activity_OpeningValve(
			index		:= E_CRYO_EVAC_VALVES_50000.PVV2, 
			nNextState	:= E_CRYO_EVAC_STATE_50000.WAIT_VAG_F_G_1);

	E_CRYO_EVAC_STATE_50000.WAIT_VAG_F_G_1:
		M_Activity_Waiting2Pressures(
			index1		:= E_CRYO_EVAC_PRESSURES_50000.VAGF, 
			index2		:= E_CRYO_EVAC_PRESSURES_50000.VAGG, 
			lrRef		:= 0.9 * cfg.lrThld_Prevac, 
			nNextState	:= E_CRYO_EVAC_STATE_50000.CLOSE_PVV2);

	E_CRYO_EVAC_STATE_50000.CLOSE_PVV2:
		M_Activity_ClosingValve(
			index		:= E_CRYO_EVAC_VALVES_50000.PVV2, 
			nNextState	:= E_CRYO_EVAC_STATE_50000.CLOSE_PVV1);

	E_CRYO_EVAC_STATE_50000.CLOSE_PVV1:
		M_Activity_ClosingValve(
			index		:= E_CRYO_EVAC_VALVES_50000.PVV1, 
			nNextState	:= E_CRYO_EVAC_STATE_50000.START_TMP);

	E_CRYO_EVAC_STATE_50000.START_TMP:
		M_Activity_StartingTMP();
		
	E_CRYO_EVAC_STATE_50000.OPEN_PVV3:
		M_Activity_OpeningValve(
			index		:= E_CRYO_EVAC_VALVES_50000.PVV3, 
			nNextState	:= E_CRYO_EVAC_STATE_50000.WAIT_VAG_2_3);

	E_CRYO_EVAC_STATE_50000.WAIT_VAG_2_3:
		M_Activity_Waiting2Pressures(
			index1		:= E_CRYO_EVAC_PRESSURES_50000.VAG2, 
			index2		:= E_CRYO_EVAC_PRESSURES_50000.VAG3, 
			lrRef		:= cfg.lrThld_Prevac, 
			nNextState	:= E_CRYO_EVAC_STATE_50000.OPEN_PVV4);

	E_CRYO_EVAC_STATE_50000.OPEN_PVV4:
		M_Activity_OpeningValve(
			index		:= E_CRYO_EVAC_VALVES_50000.PVV4, 
			nNextState	:= E_CRYO_EVAC_STATE_50000.WAIT_VAG_F_G_2);

	E_CRYO_EVAC_STATE_50000.WAIT_VAG_F_G_2:
		M_Activity_Waiting2Pressures(
			index1		:= E_CRYO_EVAC_PRESSURES_50000.VAGF, 
			index2		:= E_CRYO_EVAC_PRESSURES_50000.VAGG, 
			lrRef		:= cfg.lrThld_Vacuum, 
			nNextState	:= E_CRYO_EVAC_STATE_50000.CLOSE_GBV);

	E_CRYO_EVAC_STATE_50000.CLOSE_GBV:
		M_Activity_ClosingValve(
			index		:= E_CRYO_EVAC_VALVES_50000.GBV, 
			nNextState	:= E_CRYO_EVAC_STATE_50000.EVACUATING);

	E_CRYO_EVAC_STATE_50000.EVACUATING:
		M_Activity_Evacuating();

	E_CRYO_EVAC_STATE_50000.CLOSE_ALL_VALVES:
		M_Activity_ClosingAllValves();

	E_CRYO_EVAC_STATE_50000.DELAY_STOPPING:
		M_Activity_DelayBeforeStoppingPumps();

	E_CRYO_EVAC_STATE_50000.STOP_TMP_1:
		M_Activity_StoppingTMP(1);

	E_CRYO_EVAC_STATE_50000.STOP_PVP:
		M_Activity_StoppingPVP();

	E_CRYO_EVAC_STATE_50000.WAIT_TMP_STANDSTILL:
		M_Activity_WaitingTMP2Stop();

	E_CRYO_EVAC_STATE_50000.STOP_TMP_2:
		M_Activity_StoppingTMP(2);

	
END_CASE
END_METHOD

METHOD M_UpdateStatus
VAR_INPUT
END_VAR
stat.bEnabled		:= in_bEnable;
stat.bRootPumpON	:= rpRef.M_IsReady();
stat.bTurboPumpON	:= tpRef.M_IsReady();
END_METHOD

END_FUNCTION_BLOCK

// ---- POUs/Actuators/FB_CRYO_ACTUATOR_CMD.TcPOU
FUNCTION_BLOCK FB_CRYO_ACTUATOR_CMD
VAR_INPUT
	in_bEnable:		BOOL;			// External ON/OFF command
	in_bInterlock:	BOOL := FALSE;	// External Interlock
END_VAR
VAR_OUTPUT
	out_bEnable:	BOOL := FALSE;	// Resulting command
END_VAR
VAR
	bAutoMode:		BOOL := TRUE;	// AUTO=true, MANUAL=false
	bEngMode:		BOOL := FALSE;	// Commissioning/Engineering mode. Ignores interlocks
	
	// Disable/enable manual control buttons
	bDisableBtnOn:	BOOL := FALSE;
	bDisableBtnOff:	BOOL := FALSE;

	// ON/OFF command permissions
	bPermitOn:		BOOL := TRUE;
	bPermitOff:		BOOL := TRUE;
	
	// Handling of Manual commands
	bManualCmd:		BOOL := FALSE;
	bManualExecute:	BOOL := FALSE;
	
	// Reset interlocks (if possible)
	bReset:			BOOL := FALSE;
END_VAR

IF bAutoMode THEN
	// Simplest case, no restrictions.
	out_bEnable	:= in_bEnable;
	// Disable Manual control buttons
	bDisableBtnOn	:= TRUE;
	bDisableBtnOff	:= TRUE;
ELSIF bEngMode	THEN
	// No restrictions, no safety !!!
	// User responsible for damage caused by wrong/dangerous commands.
	IF bManualExecute THEN
		// Assign user command to the output without any checks !!!
		out_bEnable		:= bManualCmd;
		// Clear command trigger
		bManualExecute	:= FALSE;
	END_IF
	// Enable Manual control buttons
	bDisableBtnOn	:= FALSE;
	bDisableBtnOff	:= FALSE;
ELSIF NOT bAutoMode	THEN
	//
	// Manual mode.
	//
	// Only permitted commands can be executed.
	IF bManualExecute THEN
		// Execute only permitted commands.
		IF	(bManualCmd = TRUE   AND  bPermitOn)  OR
			(bManualCmd = FALSE  AND  bPermitOff) 	THEN
			// Assign user command to the output.
			out_bEnable		:= bManualCmd;
		END_IF
		// Clear command trigger
		bManualExecute	:= FALSE;
	ELSIF in_bInterlock THEN 
		// Interlock active
		IF bPermitOn AND bPermitOff THEN
			// Enable Manual control of both ON&OFF buttons
			bDisableBtnOn	:= FALSE;
			bDisableBtnOff	:= FALSE;
		ELSIF bPermitOn THEN
			// Manual Mode and only ON is permitted.
			out_bEnable		:= TRUE;
			// Enable Manual control ON button
			bDisableBtnOn	:= FALSE;
			bDisableBtnOff	:= TRUE;
		ELSIF bPermitOff THEN
			// Manual Mode and only OFF is permitted.
			out_bEnable		:= FALSE;
			// Enable Manual control OFF button
			bDisableBtnOn	:= TRUE;
			bDisableBtnOff	:= FALSE;
		END_IF
	ELSIF NOT in_bInterlock THEN
		// Enable/Disable Manual control buttons
		bDisableBtnOn	:= NOT bPermitOn;
		bDisableBtnOff	:= NOT bPermitOFF;
	END_IF
END_IF

METHOD M_SetPermissionOff
VAR_INPUT
	in_bPermit:	BOOL;
END_VAR
bPermitOff	:= in_bPermit;
END_METHOD

METHOD M_SetPermissionOn
VAR_INPUT
	in_bPermit:	BOOL;
END_VAR
bPermitOn	:= in_bPermit;
END_METHOD

METHOD M_SetPermissions
VAR_INPUT
	in_bPermitOn:	BOOL;
	in_bPermitOff:	BOOL;
END_VAR
bPermitOn	:= in_bPermitOn;
bPermitOff	:= in_bPermitOff;
END_METHOD

END_FUNCTION_BLOCK

// ---- POUs/Coolers/FB_CRYO_CRYOTELGT.TcPOU
// Cryotel GT Cooler Control
FUNCTION_BLOCK FB_CRYO_CRYOTELGT EXTENDS FB_RS_BASE
VAR_INPUT
	{attribute 'OPC.UA.DA' := '0'}
	in_bEnable:			BOOL;			// Flag to Start/Stop cooler
	{attribute 'OPC.UA.DA' := '0'}
	in_bAutoMonitor:	BOOL := TRUE;	// If true, it starts PERIODIC reads (monitoring) after INIT
	{attribute 'OPC.UA.DA' := '0'}
	in_nPeriod:			DINT := 2000;	// Interval for periodic reading [ms], default 2000 ms = 2 sec
	{attribute 'OPC.UA.DA' := '0'}
	in_sCmdSuffix:		STRING(16) := '$0D';
	{attribute 'OPC.UA.DA' := '0'}
	in_sReplySuffix:	STRING(16) := '$0D';
END_VAR
VAR_OUTPUT
END_VAR
VAR

	{attribute 'OPC.UA.DA' := '0'}
	comm:		FB_RS_COMM_CRYOTELGT;	// FB_RS_COMM_NO_SIM;		// No simulation yet
	
	// Pointers to structures inside FB_RS_COMM, e.g. ptrCommCfg.
	{attribute 'OPC.UA.DA' := '0'}
	ptrCommCfg:		POINTER TO T_RS_COMM_CFG;	(* Pointer to comm.cfg instance *)
	{attribute 'OPC.UA.DA' := '0'}
	ptrCommCtrl:	POINTER TO T_RS_COMM_CTRL;	(* Pointer to comm.ctrl instance *)
	{attribute 'OPC.UA.DA' := '0'}
	ptrCommStat:	POINTER TO T_RS_COMM_STAT;	(* Pointer to comm.stat instance *)
	
	
	{attribute 'OPC.UA.DA' := '0'}
	cfg:			T_CRYO_CRYOTELGT_CFG;	
	{attribute 'OPC.UA.DA' := '0'}
	ctrl:			T_CRYO_CRYOTELGT_CTRL;	
	{attribute 'OPC.UA.DA' := '0'}
	stat:			T_CRYO_CRYOTELGT_STAT;	

	// Pointers to arrays of INIT and READ commands
	{attribute 'OPC.UA.DA' := '0'}
	ptrInitCmds:	POINTER TO ARRAY [1..8]  OF T_CRYO_CRYOTELGT_CMD;(* Pointer to INIT commands *)
	{attribute 'OPC.UA.DA' := '0'}
	ptrReadCmds:	POINTER TO ARRAY [1..16] OF T_CRYO_CRYOTELGT_CMD;(* Pointer to READ commands *)


	(* Timers *)
	{attribute 'OPC.UA.DA' := '0'}
	fbTimer:		TON; 	// General Timeout
	timerState:		TON;	// Timer for state changes
	
	// Triggers
	triggerStart:	R_TRIG;
	triggerStop:	F_TRIG;
	

	(* Misc internal vars *)
	{attribute 'OPC.UA.DA' := '0'}
	cmdCounter:		INT := 1;	// Position in commands table
	{attribute 'OPC.UA.DA' := '0'}
	bResult:		BOOL := FALSE;
	{attribute 'OPC.UA.DA' := '0'}
	bStarted:		BOOL := FALSE;

	// TODO: Add Input signals in Fbs that EXTEND this FB.

	// Output signals
	q_bStart		AT %Q*:	BOOL;	// Start/Stop the cooler. Common to all.



END_VAR

// Hard-coded configuration
M_Configure();

(* Execute comm instance *)
M_ExecuteComm();
//comm(in_sCmdSuffix:=in_sCmdSuffix, in_sReplySuffix:=in_sReplySuffix, in_nTimeout:=3000);

// Update cooler status from digital signals.
M_UpdateStatus();

// Capture Start/Stop commands and execute the State Machine
M_StateMachine();

// Execute the base class object FB_RS_BASE
SUPER^();

METHOD ActivityInitializing
VAR_INPUT
	bExecute:	BOOL;
END_VAR
VAR_INST
	{attribute 'OPC.UA.DA' := '0'}
    nMethodState:	INT := 0;	// State Machine current state
END_VAR
VAR
	bReadOK:	BOOL;
END_VAR
SetAction('ActivityInitializing');


IF NOT bExecute THEN
	nMethodState	:= 0;	// Reset the state machine
	cmdCounter		:= 0;	// Init will start from the first init command after increment
	RETURN;
END_IF

// Handle State Machine
CASE nMethodState OF
	0:	// Set initial state and status
		stat.bInitialised	:= FALSE;
		stat.sReply			:= '';
		SetStatus(E_SM_ERROR.OK, 'BUSY');

		nMethodState := 10;				// Go to next state, i.e. INIT_COMM

	10:	// Initialize COMM port
		(* Reset the serial port *)
		ptrCommCtrl^.nCommand	:= E_RS_COMM_CMD.INIT;
		ptrCommCtrl^.bExecute	:= TRUE;

		(* Start the timer by going false/true *)
		fbTimer (IN := FALSE); (* Reset timer *)
		fbTimer (IN := TRUE, PT := T#5S); (* 5 sec timeout for reply *)

		nMethodState 	:= 15;	// On next cycle wait until the comm port is reset, i.e. idle
		
	15:	// Wait IDLE
		fbTimer (IN := TRUE);
		IF comm.stat.nStatus = E_RS_COMM_STATUS.IDLE THEN
			// Communication is IDLE 
			fbTimer (IN := FALSE);	// disable timer 
			stat.sReply		:= ptrCommStat^.sReply;	// Save the reply

			// Read from the reply.
			// Argument TRUE means that this is an INIT command.
			bReadOK	:= M_ReadFromReply(cmdCounter, TRUE);
			IF NOT bReadOK	THEN
				cmdCounter		:= 0;	// Reset command counter
				nMethodState 	:= 10;	// Wait for INIT
			ELSE
				cmdCounter		:= cmdCounter + 1;	// Increment init command index
				fbTimer (IN := FALSE);	// disable timer 
				fbTimer (IN := TRUE, PT := cfgRef.tDelay_Init); // Wait INIT delay
				bCommProblem	:= FALSE;
				nMethodState 	:= 18;	// Execute next device INIT command
			END_IF
		ELSIF comm.stat.nStatus = E_RS_COMM_STATUS.ERROR THEN
			fbTimer (IN := FALSE);
			SetStatus(E_LAKESHORE_ERROR.COMM, 'ERROR: Communication error');	
			bCommProblem	:= TRUE;
			nEvent := E_SM_EVENT.ERRINIT;
			RETURN;
		ELSIF fbTimer.Q THEN
			// Timer expired after 5 sec. This is an error.
			fbTimer (IN := FALSE);
			SetStatus(E_LAKESHORE_ERROR.TIMEOUT, 'ERROR: Communication timeout');	
			bCommProblem	:= TRUE;
			nEvent := E_SM_EVENT.ERRINIT;
			RETURN;
		END_IF

	
	
	18:	// Wait INIT Delay
		fbTimer (IN := TRUE);
		IF fbTimer.Q THEN
			// Timer expired after 5 sec. This is an error.
			fbTimer (IN := FALSE);
			nMethodState 	:= 20;	// Execute next device INIT command
			RETURN;
		END_IF

	
	
	20:	// INIT DEV
		IF ptrInitCmds^ [cmdCounter].cmd = '' THEN
			// Device INIT is done. Go to IDLE 
			stat.bInitialised 	:= TRUE;
			cmdCounter			:= 1;
			SetStatus(E_SM_ERROR.OK, 'IDLE');
			nEvent 		:= E_SM_EVENT.INITDONE;
			RETURN;
		END_IF
		
		(* Send INIT command with index cmdCounter *)
		ptrCommCtrl^.nCommand		:= E_RS_COMM_CMD.SEND;
		ptrCommCtrl^.sCmd			:= ptrInitCmds^ [cmdCounter].cmd;
		ptrCommCtrl^.nNumReplies	:= ptrInitCmds^ [cmdCounter].nReplies;
		ptrCommCtrl^.bHasReply		:= ptrInitCmds^ [cmdCounter].nReplies > 0;
		ptrCommCtrl^.bExecute		:= TRUE;
	
		(* Start the timer by going false/true *)
		fbTimer (IN := FALSE); (* Reset timer *)
		fbTimer (IN := TRUE, PT := T#5S); (* 5 sec timeout for reply *)

		// On next cycle wait until the comm port is idle
		nMethodState 	:= 15;	// On next cycle wait until the comm port is idle
	
END_CASE
END_METHOD

METHOD ActivityInitializing_new
VAR_INPUT
	bExecute:	BOOL;
END_VAR
VAR_INST
	{attribute 'OPC.UA.DA' := '0'}
    nMethodState:	INT := 0;	// State Machine current state
	{attribute 'OPC.UA.DA' := '0'}
	bCommInit:		BOOL;
END_VAR
VAR
	bReadOK:	BOOL;
END_VAR
SetAction('ActivityInitializing');


IF NOT bExecute THEN
	nMethodState	:= 0;	// Reset the state machine
	cmdCounter		:= 0;	// Init will start from the first init command after increment
	RETURN;
END_IF

// Handle State Machine
CASE nMethodState OF
	0:	// Set initial state and status
		stat.bInitialised	:= FALSE;
		stat.sReply			:= '';
		SetStatus(E_SM_ERROR.OK, 'BUSY');

		nMethodState := 10;				// Go to next state, i.e. INIT_COMM

	10:	// Initialize COMM port
		(* Reset the serial port *)
		ptrCommCtrl^.nCommand	:= E_RS_COMM_CMD.INIT;
		ptrCommCtrl^.bExecute	:= TRUE;

		(* Start the timer by going false/true *)
		fbTimer (IN := FALSE); (* Reset timer *)
		fbTimer (IN := TRUE, PT := T#5S); (* 5 sec timeout for reply *)

		bCommInit		:= TRUE;
		nMethodState 	:= 15;	// On next cycle wait until the comm port is reset, i.e. idle
		
	15:	// Wait IDLE
		fbTimer (IN := TRUE);
		IF comm.stat.nStatus = E_RS_COMM_STATUS.IDLE THEN
			// If we have just executed the COMM Reset/INIT command,
			// Go to first INIT command.
			IF bCommInit THEN
				bCommInit		:= FALSE;
				cmdCounter		:= 1;	// Start from first INIT command
				fbTimer (IN := FALSE);	// disable timer 
				fbTimer (IN := TRUE, PT := cfgRef.tDelay_Init); // Wait INIT delay
				bCommProblem	:= FALSE;
				nMethodState 	:= 18;	// Execute next device INIT command
				RETURN;
			END_IF
			// Communication is IDLE 
			fbTimer (IN := FALSE);	// disable timer 
			stat.sReply		:= ptrCommStat^.sReply;	// Save the reply

			// Read from the reply.
			// Argument TRUE means that this is an INIT command.
			bReadOK	:= M_ReadFromReply(cmdCounter, TRUE);
			IF NOT bReadOK	THEN
				cmdCounter		:= 0;	// Reset command counter
				nMethodState 	:= 10;	// Wait for INIT
			ELSE
				cmdCounter		:= cmdCounter + 1;	// Increment init command index
				fbTimer (IN := FALSE);	// disable timer 
				fbTimer (IN := TRUE, PT := cfgRef.tDelay_Init); // Wait INIT delay
				bCommProblem	:= FALSE;
				nMethodState 	:= 18;	// Execute next device INIT command
			END_IF
		ELSIF comm.stat.nStatus = E_RS_COMM_STATUS.ERROR THEN
			fbTimer (IN := FALSE);
			SetStatus(E_LAKESHORE_ERROR.COMM, 'ERROR: Communication error');	
			bCommProblem	:= TRUE;
			nEvent := E_SM_EVENT.ERRINIT;
			RETURN;
		ELSIF fbTimer.Q THEN
			// Timer expired after 5 sec. This is an error.
			fbTimer (IN := FALSE);
			SetStatus(E_LAKESHORE_ERROR.TIMEOUT, 'ERROR: Communication timeout');	
			bCommProblem	:= TRUE;
			nEvent := E_SM_EVENT.ERRINIT;
			RETURN;
		END_IF

	
	
	16:	// Delay and then goto Wait for IDLE
		fbTimer (IN := TRUE);

		IF fbTimer.Q THEN
			fbTimer (IN := FALSE); // Reset timer
			fbTimer (IN := TRUE, PT := T#5S);	// 5sec timeout for reply.	
			nMethodState 	:= 15;	// Goto Wait for IDLE
			RETURN;
		END_IF
	
	18:	// Delay and then goto execute next command
		fbTimer (IN := TRUE);
		IF fbTimer.Q THEN
			// Timer expired after 5 sec. This is an error.
			fbTimer (IN := FALSE);
			nMethodState 	:= 20;	// Goto next INIT command
			RETURN;
		END_IF

	
	
	20:	// INIT DEV
		IF ptrInitCmds^ [cmdCounter].cmd = '' THEN
			// Device INIT is done. Go to IDLE 
			stat.bInitialised 	:= TRUE;
			cmdCounter			:= 1;
			SetStatus(E_SM_ERROR.OK, 'IDLE');
			nEvent 		:= E_SM_EVENT.INITDONE;
			RETURN;
		END_IF
		
		(* Send INIT command with index cmdCounter *)
		ptrCommCtrl^.nCommand		:= E_RS_COMM_CMD.SEND;
		ptrCommCtrl^.sCmd			:= ptrInitCmds^ [cmdCounter].cmd;
		ptrCommCtrl^.nNumReplies	:= ptrInitCmds^ [cmdCounter].nReplies;
		ptrCommCtrl^.bHasReply		:= ptrInitCmds^ [cmdCounter].nReplies > 0;
		ptrCommCtrl^.bExecute		:= TRUE;
	
		// In case this is a command without a reply,
		// we apply 200ms delay between commmands.
		IF NOT ptrCommCtrl^.bHasReply THEN
			// There is no reply, i.e. this is a 'SET' command.
			// Start the timer by going false/true.
			// Apply 200ms delay between SET commands.
			fbTimer (IN := FALSE); // Reset timer
			fbTimer (IN := TRUE, PT := T#200MS); 
			cmdCounter		:= cmdCounter + 1;	// Go to next command.
			nMethodState	:= 18;				// Goto WAIT for delay.
			RETURN;
		ELSE			
			// There is a reply.
			// Apply a delay of 20ms before checking the status. 
			// Start the timer by going false/true
			fbTimer (IN := FALSE); // Reset timer
			fbTimer (IN := TRUE, PT := T#5MS);	
			stat.sErrorText	:= 'BUSY';
			nMethodState := 16;	// Goto WAIT for Reading to complete,
		END_IF
		
END_CASE
END_METHOD

METHOD ActivityMonitoring
VAR_INPUT
	bExecute:	BOOL;
END_VAR
VAR_INST
	{attribute 'OPC.UA.DA' := '0'}
    nMethodState:	INT := 0;	// State Machine current state
	{attribute 'OPC.UA.DA' := '0'}
	nRetries:		INT := 0;	// Number of retries in case of communication problems
END_VAR

VAR
	offset: INT;
	bReadOK:	BOOL;
END_VAR
IF NOT cfgRef.bAutoMonitor AND stat.nSubstate = E_RS_BASE_SUBSTATE.NOTOP_READY THEN
	SetAction('No Monitoring'); 
	SetStatus(E_SM_ERROR.OK, 'IDLE');
	nMethodState	:= 0;	// Reset the state machine
	cmdCounter		:= 1;	// Reading will start from the first command in the array
	RETURN;
END_IF

IF NOT bExecute THEN
	SetAction('ActivityMonitoring'); 
	SetStatus(E_SM_ERROR.OK, 'BUSY');
	nMethodState	:= 0;	// Reset the state machine
	cmdCounter		:= 1;	// Reading will start from the first command in the array
	RETURN;
END_IF

// Handle State Machine
CASE nMethodState OF
	0:	// Execute a command from the command array
		IF ptrReadCmds^ [cmdCounter].cmd = '' OR cmdCounter > 16 THEN

			// All commands have been executed. 
			// Wait tDelay_Periodic before re-starting the READ.
			cmdCounter	:= 1;
			SetStatus(E_SM_ERROR.OK, 'IDLE');
			
			(* Start the timer by going false/true *)
			fbTimer (IN := FALSE); (* Reset timer *)
			fbTimer (IN := TRUE, PT := cfgRef.tDelay_Periodic);
			nMethodState := 10;				// Goto Wait for tDelay_Periodic
			RETURN;
			
		END_IF
		
		(* Send command with index cmdCounter *)
		ptrCommCtrl^.nCommand		:= E_RS_COMM_CMD.SEND;
		ptrCommCtrl^.sCmd			:= ptrReadCmds^ [cmdCounter].cmd;
		ptrCommCtrl^.nNumReplies	:= ptrReadCmds^ [cmdCounter].nReplies;
		ptrCommCtrl^.bHasReply		:= ptrReadCmds^ [cmdCounter].nReplies > 0;
		ptrCommCtrl^.bExecute		:= TRUE;
		
		// In case we are executing 'SET' commands, there are no replies.
		// However, we need a delay of at least 50ms between commands.
		// We will apply 150ms.
		IF NOT ptrCommCtrl^.bHasReply THEN
			// There is no reply, i.e. this is a 'SET' command.
			// Start the timer by going false/true.
			// Apply 200ms delay between SET commands.
			fbTimer (IN := FALSE); // Reset timer
			fbTimer (IN := TRUE, PT := T#200MS); 
			cmdCounter		:= cmdCounter + 1;	// Go to next command.
			nMethodState	:= 10;				// Goto WAIT for Reading to complete,
			RETURN;
		ELSE			
			// There is a reply, i.e. this is a 'READ' command.
			// Apply a delay of 10ms before checking the status. 
			// Start the timer by going false/true
			fbTimer (IN := FALSE); // Reset timer
			fbTimer (IN := TRUE, PT := T#10MS);	
			stat.sErrorText	:= 'BUSY';
			nMethodState := 15;	// Goto WAIT for Reading to complete,
		END_IF
		

	10:	// Wait until the delay timeout expires
		fbTimer (IN := TRUE);

		(* If Timer has expired, go to the next state. *)
		IF fbTimer.Q THEN
			fbTimer (IN := FALSE);
			nMethodState 	:= 0;	// Goto Wait for tDelay_Periodic
			RETURN;
		END_IF
	
	15:	// Wait until the delay timeout expires
		fbTimer (IN := TRUE);

		(* If Timer has expired, go to the next state. *)
		IF fbTimer.Q THEN
			fbTimer (IN := FALSE);
			fbTimer (IN := TRUE, PT := T#5S);	// 5 sec timeout for reply
			stat.sErrorText	:= 'BUSY';
			nMethodState 	:= 20;	// Goto Wait for IDLE/Reply
			RETURN;
		END_IF
	



	20:	// Wait for the reading to complete, i.e. IDLE
		fbTimer (IN := TRUE);
		IF comm.stat.nStatus = E_RS_COMM_STATUS.IDLE THEN
			// Communication is IDLE 
			fbTimer (IN := FALSE);	// disable timer 
			stat.sReply		:= ptrCommStat^.sReply;	// Save the reply
			
			// Copy readings to status variable(s)
			
			// Read from the reply.
			// Argument FALSE means that this is NOT an INIT command.
			bReadOK	:= M_ReadFromReply(cmdCounter, FALSE);
			IF NOT bReadOK	THEN
				// Reply was not OK. Maybe out of sync.
				// Re-INIT the communication, i.e. clear the buffer.
				ptrCommCtrl^.nCommand	:= E_RS_COMM_CMD.INIT;
				ptrCommCtrl^.bExecute	:= TRUE;
		
				(* Start the timer by going false/true *)
				fbTimer (IN := FALSE); (* Reset timer *)
				fbTimer (IN := TRUE, PT := T#5S); (* 5 sec timeout for reply *)
		
				SetStatus(E_LAKESHORE_ERROR.COMM, 'ERROR: Communication error');	
				bCommProblem	:= TRUE;

				nMethodState 	:= 10;	// On next cycle wait until the comm port is reset, i.e. idle
				RETURN;
			ELSE
				// All OK. Go to next command.
				bCommProblem	:= FALSE;
				nRetries		:= 0;	// Reset number of retries
		
				cmdCounter		:= cmdCounter + 1;	// Go to next command.
				
				// Apply a 150 ms delay between commands
				fbTimer (IN := FALSE);	// Reset timer
				fbTimer (IN := TRUE, PT := cfg.tDelay_Read); 
				nMethodState := 10;		// Apply delay
				nEvent := E_SM_EVENT.COMMOK;
				RETURN;
			END_IF
		ELSIF comm.stat.nStatus = E_RS_COMM_STATUS.ERROR OR fbTimer.Q THEN
			// No Reply.
			// Re-INIT the communication, i.e. clear the buffer.
			ptrCommCtrl^.nCommand	:= E_RS_COMM_CMD.INIT;
			ptrCommCtrl^.bExecute	:= TRUE;
	
			(* Start the timer by going false/true *)
			fbTimer (IN := FALSE); (* Reset timer *)
			fbTimer (IN := TRUE, PT := T#5S); (* 5 sec timeout for reply *)
	
			SetStatus(E_LAKESHORE_ERROR.COMM, 'ERROR: Communication error');	
			bCommProblem	:= TRUE;

			nRetries		:= nRetries + 1;		// Increment number of retries
			stat.nRetries	:= stat.nRetries + 1;	// Increment total number of retries

			nMethodState 	:= 10;	// On next cycle wait until the comm port is reset, i.e. idle
			RETURN;
		END_IF

	
END_CASE
END_METHOD

METHOD M_AddCtrlCommands : BOOL
VAR_INPUT
//	in_sCmd:	STRING;
END_VAR
VAR
	i:	INT;
    fbFormat:	FB_FormatString;
	nVal:		UDINT;
	lrVal:		LREAL;
	sPowerCmd:	STRING;
END_VAR
// Find index of first two empty commands.
// The result must be greater than zero, if everuthing is OK.
i	:= M_FindReadCommand('');

// Add relevant control commands to the end of the list
// of Read/status comands.
IF i > 0	THEN
	IF ctrl.nDevCmd	= E_CRYO_CRYOTELGT_CMD.ON	THEN
		// Cooler is always started with 240W output.
		// Write the output power and then the ON command.
		ctrl.lrPower	:= 240.0;
		cfg.cmdList_Read[i].cmd			:= 'PWOUT=240';
		cfg.cmdList_Read[i+1].cmd		:= 'COOLER=POWER';
		// Each command has a single reply.
		cfg.cmdList_Read[i].nReplies	:= 2;
		cfg.cmdList_Read[i+1].nReplies	:= 2;
	ELSIF ctrl.nDevCmd	= E_CRYO_CRYOTELGT_CMD.OFF	THEN
		// Write the power OFF command.
		cfg.cmdList_Read[i].cmd			:= 'COOLER=OFF';
		cfg.cmdList_Read[i+1].cmd		:= '';
		// Each command has a single reply.
		cfg.cmdList_Read[i].nReplies	:= 2;
		cfg.cmdList_Read[i+1].nReplies	:= 0;
	ELSIF ctrl.nDevCmd	= E_CRYO_CRYOTELGT_CMD.SET_POWER	THEN
		// Updating only the power value.
		ctrl.bPower	:= TRUE;
		// Write the output power command.
		lrVal	:= ctrl.lrPower;
		fbFormat(	sFormat := 'PWOUT=%.2f', 
					arg1 := F_LREAL(lrVal), 
					sOut => sPowerCmd);
		cfg.cmdList_Read[i].cmd			:= sPowerCmd;
		cfg.cmdList_Read[i+1].cmd		:= '';
		// Each command has a single reply.
		cfg.cmdList_Read[i].nReplies	:= 2;
		cfg.cmdList_Read[i+1].nReplies	:= 0;
	END_IF
	
	M_AddCtrlCommands	:= TRUE;
ELSE
	M_AddCtrlCommands	:= FALSE;
END_IF
END_METHOD

METHOD M_ClearCtrlCommands
VAR_INPUT
END_VAR
VAR
	i:	INT;
END_VAR
// Search for commands starting with  'COOLER=' and 'PWOUT='.
// If found, clear them.
FOR i := 1 TO 16 DO
	IF FIND(cfg.cmdList_Read[i].cmd, 'PWOUT=') > 0	THEN
		cfg.cmdList_Read[i].cmd	:= '';
	ELSIF FIND(cfg.cmdList_Read[i].cmd, 'COOLER=') > 0	THEN
		cfg.cmdList_Read[i].cmd	:= '';
	END_IF
END_FOR

ctrl.nDevCmd	:= E_CRYO_CRYOTELGT_CMD.NONE;
ctrl.bPower		:= FALSE;
END_METHOD

METHOD M_Configure
VAR_INPUT
END_VAR
VAR
		i:	INT;
END_VAR
IF NOT bStarted	THEN
	//
	// START: Mandatory  !!!
	//
	// Set references from FB_RS_BASE
	cfgRef	REF=cfg;
	ctrlRef	REF=ctrl;
	statRef	REF=stat;

	// Ensure that the references are correctly set
	IF	NOT __ISVALIDREF(cfgRef)	OR  
		NOT __ISVALIDREF(ctrlRef)	OR  
		NOT __ISVALIDREF(statRef)		THEN
		stat.sErrorText	:= 'References not configured';
		RETURN;
	END_IF
	
	// Copy input parameters to configuration
	cfg.bAutoMonitor	:= in_bAutoMonitor;
	cfg.tDelay_Periodic	:= DINT_TO_TIME(in_nPeriod);
	cfg.tDelay_Ctrl		:= T#200MS;
	
	
	// Set pointers to arrays of commands
	ptrInitCmds	:= ADR(cfg.cmdList_Init);(* Pointer to INIT commands *)
	ptrReadCmds	:= ADR(cfg.cmdList_Read);(* Pointer to READ commands *)
	
	// TODO in FB that extends the functionality
	// Set pointers to comm, i.e.
	ptrCommCfg	:= ADR(comm.cfg);	(* Pointer to comm.cfg instance *)
	ptrCommCtrl	:= ADR(comm.ctrl);	(* Pointer to comm.ctrl instance *)
	ptrCommStat	:= ADR(comm.stat);	(* Pointer to comm.stat instance *)
	
	// Set comm suffixes for commands and replies
	ptrCommCfg^.sCmdSuffix		:= in_sCmdSuffix;
	ptrCommCfg^.sReplySuffix	:= in_sReplySuffix;

	stat.bConfigured	:= TRUE;
	bStarted			:= TRUE;
	//
	// END: Mandatory for ALL cooler !!!
	//


	
END_IF
END_METHOD

METHOD M_ExecuteComm
VAR_INPUT
END_VAR
comm(	in_bSimulation	:= in_bSimulation, 
		in_sCmdSuffix	:= in_sCmdSuffix, 
		in_sReplySuffix	:= in_sReplySuffix, 
		in_nTimeout		:= 3000);
END_METHOD

// Return the index of the command in cfg.cmdList_Read[].
// Returns zero if not found.
METHOD M_FindReadCommand : INT
VAR_INPUT
	in_sCmd:	STRING;
END_VAR
VAR
	i:	INT;
END_VAR
// We need two empty commands: 'COOLER=<>' and 'PWOUT=<VAL>'.
// Thats's why the highest index is 15 rather than 16.
FOR i := 1 TO 15 DO
	IF cfg.cmdList_Read[i].cmd = in_sCmd	THEN
		M_FindReadCommand	:= i;
		RETURN;
	END_IF
END_FOR

M_FindReadCommand	:= 0;
END_METHOD

METHOD M_GetCouplerState : BOOL
VAR_INPUT
END_VAR
IF comm.i_nCouplerState = 8  OR  comm.in_bSimulation  THEN
	M_GetCouplerState	:= TRUE;	
ELSE
	M_GetCouplerState	:= FALSE;	
END_IF
END_METHOD

METHOD M_ReadFromReply : BOOL
// Method to check correctness of the reply and assign the result to a status variable.
VAR_INPUT
	idx:		INT;			// Command index in the array.
	bInitCmd:	BOOL := FALSE;	// If TRUE, this is an INIT command, otherwise it is Read/status
END_VAR
VAR
	pos:	INT;
	length:	INT;
	cmd:	STRING;
	subStr:	STRING;
END_VAR
// During INIT it might happen that the command index is 0.
// These cases should be discarded.
IF idx <= 0	THEN
	M_ReadFromReply	:= TRUE;
	RETURN;
END_IF

// Get the command
IF bInitCmd	THEN
	cmd		:= cfg.cmdList_Init[idx].cmd;
ELSE
	cmd		:= cfg.cmdList_Read[idx].cmd;
END_IF

// The sent command has to be included in the first line of the reply.
// If not, we are out of sync and have to reinitialise.
IF FIND(stat.sReply, cmd) = 0	THEN
	bCommProblem	:= TRUE;
	stat.nState		:= E_RS_BASE_STATE.NOTOP;
	stat.nSubstate	:= E_RS_BASE_SUBSTATE.NOTOP_NOTREADY;
	RETURN;
END_IF

// Extract the value from the reply.
// Example: 
//    Command: VERSION
//    Reply:   VERSION$R$Nv1.4.1$R
//    Value:   v1.4.1
//
// Take the string after the '$R$N' and remove the '$R' at the end.
// Remove the <CR> suffix from the reply.

pos	:= FIND(stat.sReply,'$R$N');
IF pos = 0	THEN
	// The string is not found. 
	M_ReadFromReply	:= FALSE;
	RETURN;
END_IF

length	:= LEN(stat.sReply) - pos -2;
subStr	:= MID(stat.sReply, length, pos+2);


IF cmd = 'VERSION'	THEN
	stat.sVersion	:= subStr;
ELSIF cmd = 'MODE'	THEN
	stat.sMode		:= subStr;
ELSIF cmd = 'SENSOR'	THEN
	stat.sSensor	:= subStr;
ELSIF FIND(cmd, 'PWOUT=') = 1	THEN
	// Get the commanded power from the command.
	// Get the value after the 'PWOUT=' substring.
	stat.lrPowerCommanded	:= STRING_TO_LREAL(subStr);
	// If we are updating only the power value,
	// this is then the last control command.
	IF ctrl.bPower	THEN
		// Clear the control commands from the list.
		M_ClearCtrlCommands();
		ctrl.bPower	:= FALSE;
		// Power output command is not active any more.
		stat.bPowerCmdActive	:= FALSE;
	END_IF
ELSIF FIND(cmd, 'COOLER=') = 1	THEN
	// Get the control mode 'POWER' or 'OFF'.
	stat.sCtrlMode	:= subStr;
	// This is the last control command when switching cool on/off.
	// Clear the control commands from the list.
	M_ClearCtrlCommands();
	// Power output command is not active any more.
	stat.bPowerCmdActive	:= FALSE;
ELSIF cmd = 'ERROR'	THEN
	IF FIND(subStr, '00000001') = 1	THEN
		stat.sCtrlError	:= 'High Reject Temperature';
	ELSIF FIND(subStr, '00000010') = 1	THEN
		stat.sCtrlError	:= 'Low Reject Temperature';
	ELSIF FIND(subStr, '10000000') = 1	THEN
		stat.sCtrlError	:= 'Over Current Error';
	ELSIF FIND(subStr, '11111111') = 1	THEN
		stat.sCtrlError	:= 'Invalid Configuration';
	ELSE
		stat.sCtrlError	:= 'OK';
	END_IF
ELSIF cmd = 'COOLER'	THEN
	stat.sCtrlMode	:= subStr;
ELSIF cmd = 'P'	THEN
	stat.lrPowerMeasured	:= STRING_TO_LREAL(subStr);
ELSIF cmd = 'PWOUT'	THEN
	stat.lrPowerCommanded	:= STRING_TO_LREAL(subStr);
ELSIF cmd = 'TC'	THEN
	stat.lrTempColdHead		:= STRING_TO_LREAL(subStr);
ELSIF cmd = 'TEMP RJ'	THEN
	stat.lrTempReject		:= STRING_TO_LREAL(subStr);
ELSIF cmd = 'TTARGET'	THEN
	stat.lrTempTarget		:= STRING_TO_LREAL(subStr);
END_IF


M_ReadFromReply	:= TRUE;	// OK
END_METHOD

METHOD M_StateMachine
VAR_INPUT
END_VAR
//////////////////////
// Cooler State Machine
//////////////////////
CASE stat.nDevState OF
	E_CRYO_CRYOTELGT_STATE.OFF:
		// Capture START command when in_bEnable goes TRUE.
		triggerStart(CLK:=in_bEnable);
		IF triggerStart.Q	THEN
			// in_bEnable is TRUE, start the cooler.
			ctrl.bStart		:= TRUE;	// For digital control. Not used currently.
			ctrl.nDevCmd	:= E_CRYO_CRYOTELGT_CMD.ON;
			M_AddCtrlCommands();	// Add ON related commands
			stat.nDevState	:= 	E_CRYO_CRYOTELGT_STATE.STARTING;
			stat.sDevState	:= 'Starting...';
			// Restart the timer
			timerState(IN:=FALSE);
			timerState(IN:=TRUE,PT:=UDINT_TO_TIME(cfg.nTimeoutState));
		END_IF
	E_CRYO_CRYOTELGT_STATE.STARTING:
		timerState();	// Timeout for the state transition.
		triggerStop(CLK:= in_bEnable);	// Check if the cooler should be switched OFF.
		IF timerState.Q THEN
			// Timeout, stop the cooler.
			ctrl.bStart		:= FALSE;
			timerState(IN:=FALSE);
			M_ClearCtrlCommands();	// Clear ON related commands
			stat.nDevState	:= 	E_CRYO_CRYOTELGT_STATE.ERROR;
			stat.sDevState	:= 'ERROR - Timeout on START';
		ELSIF stat.sCtrlMode = 'POWER' THEN
			// State is 'POWER'.
			// That means that the cooler is ON in power mode.
			timerState(IN:=FALSE);
			M_ClearCtrlCommands();	// Clear ON related commands
			stat.nDevState	:= 	E_CRYO_CRYOTELGT_STATE.ON;
			stat.sDevState	:= 'ON';
		ELSIF triggerStop.Q THEN
			// in_bEnable is FALSE, stop the cooler.
			ctrl.bStart		:= FALSE;
			ctrl.nDevCmd	:= E_CRYO_CRYOTELGT_CMD.OFF;
			ctrl.lrPower	:= 240.0;
			M_ClearCtrlCommands();	// Clear ON related commands
			M_AddCtrlCommands();	// Add OFF related commands
			// Restart the timer
			timerState(IN:=FALSE);
			timerState(IN:=TRUE,PT:=UDINT_TO_TIME(cfg.nTimeoutState));
			stat.nDevState	:= 	E_CRYO_CRYOTELGT_STATE.STOPPING;
			stat.sDevState	:= 'Stopping...';
		END_IF
	E_CRYO_CRYOTELGT_STATE.ON:
		triggerStop(CLK:= in_bEnable);
		IF triggerStop.Q THEN
			// in_bEnable is FALSE, stop the cooler.
			// Restart the timer for state transition.
			ctrl.bStart		:= FALSE;
			ctrl.nDevCmd	:= E_CRYO_CRYOTELGT_CMD.OFF;
			M_AddCtrlCommands();	// Add OFF related commands
			timerState(IN:=FALSE);
			timerState(IN:=TRUE,PT:=UDINT_TO_TIME(cfg.nTimeoutState));
			stat.nDevState	:= 	E_CRYO_CRYOTELGT_STATE.STOPPING;
			stat.sDevState	:= 'Stopping...';
		ELSIF stat.sCtrlMode <> 'POWER' THEN
			// 'POWER' is the only operational mode.
			// If it is something else, stop the cooler.
			ctrl.bStart		:= FALSE;
			ctrl.nDevCmd	:= E_CRYO_CRYOTELGT_CMD.OFF;
			M_AddCtrlCommands();	// Add OFF related commands
			stat.nDevState	:= 	E_CRYO_CRYOTELGT_STATE.ERROR;
			stat.sDevState	:= 'ERROR - Unexpected OFF';
		ELSIF stat.lrTempColdHead < 100.0  AND ctrl.lrPower < 250.0	THEN
			// Switch the power to 250W if the cold head temperature is below 100K.
			IF NOT stat.bPowerCmdActive	THEN
				stat.bPowerCmdActive	:= TRUE;
				ctrl.lrPower			:= 250.0;
				ctrl.nDevCmd			:= E_CRYO_CRYOTELGT_CMD.SET_POWER;
				M_AddCtrlCommands();	// Add OFF related commands
			END_IF
		ELSIF stat.lrTempColdHead > 101.0  AND ctrl.lrPower > 240.0	THEN
			// Switch the power to 240W if the cold head temperature is above 101K.
			IF NOT stat.bPowerCmdActive	THEN
				stat.bPowerCmdActive	:= TRUE;
				ctrl.lrPower			:= 240.0;
				ctrl.nDevCmd			:= E_CRYO_CRYOTELGT_CMD.SET_POWER;
				M_AddCtrlCommands();	// Add OFF related commands
			END_IF
		END_IF
	E_CRYO_CRYOTELGT_STATE.STOPPING:
		timerState();
		// Capture START command
		triggerStart(CLK:=in_bEnable);
		IF timerState.Q THEN
			timerState(IN:=FALSE);
			M_ClearCtrlCommands();	// Clear OFF related commands
			stat.nDevState	:= 	E_CRYO_CRYOTELGT_STATE.ERROR;
			stat.sDevState	:= 'ERROR - Timeout on STOP';
		ELSIF stat.sCtrlMode = 'OFF' THEN
			timerState(IN:=FALSE);
			M_ClearCtrlCommands();	// Clear OFF related commands
			stat.nDevState	:= 	E_CRYO_CRYOTELGT_STATE.OFF;
			stat.sDevState	:= 'OFF';
		ELSIF triggerStart.Q THEN
			// in_bEnable is TRUE, start the cooler.
			ctrl.bStart		:= TRUE;
			M_ClearCtrlCommands();	// Clear OFF related commands
			ctrl.nDevCmd	:= E_CRYO_CRYOTELGT_CMD.ON;
			M_AddCtrlCommands();	// Add ON related commands
			stat.nDevState	:= 	E_CRYO_CRYOTELGT_STATE.STARTING;
			stat.sDevState	:= 'Starting...';
			// Restart the timer
			timerState(IN:=FALSE);
			timerState(IN:=TRUE,PT:=UDINT_TO_TIME(cfg.nTimeoutState));
		END_IF
	E_CRYO_CRYOTELGT_STATE.ERROR:
		// To recover from error, STOP command has to be issued
		// in order to reset triggerStop.
		// Capture STOP command
		triggerStop(CLK:=in_bEnable);
		IF triggerStop.Q THEN
			// in_bEnable is FALSE, stop the cooler.
			ctrl.nDevCmd	:= E_CRYO_CRYOTELGT_CMD.OFF;
			M_AddCtrlCommands();	// Add ON related commands
			stat.nDevState	:= 	E_CRYO_CRYOTELGT_STATE.STOPPING;
			stat.sDevState	:= 'OFF';
			RETURN;
		END_IF
		
		// Capture START command.
		triggerStart(CLK:=in_bEnable);
		IF triggerStart.Q THEN
			// in_bEnable is TRUE, start the cooler.
			ctrl.bStart		:= TRUE;
			ctrl.nDevCmd	:= E_CRYO_CRYOTELGT_CMD.ON;
			M_AddCtrlCommands();	// Add ON related commands
			stat.nDevState	:= 	E_CRYO_CRYOTELGT_STATE.STARTING;
			stat.sDevState	:= 'Starting...';
			// Restart the timer
			timerState(IN:=FALSE);
			timerState(IN:=TRUE,PT:=UDINT_TO_TIME(cfg.nTimeoutState));
		END_IF
END_CASE


// Update outputs
q_bStart	:= ctrl.bStart;
END_METHOD

METHOD M_UpdateStatus
VAR_INPUT
END_VAR
// TODO: For each cooler FB that extends FB_CRYO_PUMP_BASE update inputs in M_UpdateStatus(), e.g.

(*
// Update inputs
stat.bReady		:= i_bReady;
stat.bSpeed100	:= i_bSpeed100;
stat.bWarning	:= i_bWarning;
stat.bAlarm		:= i_bAlarm;

CASE stat.nCtrlMode	OF
	0:	stat.sCtrlMode	:= 'HHR (Hand-Held Remote)';
	1:	stat.sCtrlMode	:= 'REMOTE';
	2:	stat.sCtrlMode	:= 'SERIAL LINK';
	3:	stat.sCtrlMode	:= 'FIELDBUS';
ELSE
	stat.sCtrlMode	:= 'UNKNOWN';
END_CASE

*)
END_METHOD

METHOD ProcessEvents
VAR_INPUT
END_VAR

(* 
	Before processing the event, execute the Do-Activity tasks. 
	Note that, in case of orthogonal regions, more than one Do-Activity 
	could run in the same PLC cycle.
	Note: Most of these activities have timeouts since they take time.
*)

IF	statRef.nSubstate = E_RS_BASE_SUBSTATE.OP_MONITORING 		OR 
	statRef.nSubstate = E_RS_BASE_SUBSTATE.NOTOP_READY			OR
	(statRef.nSubstate = E_RS_BASE_SUBSTATE.NOTOP_ERROR 	AND 
	 nLastGoodSubstate = E_RS_BASE_SUBSTATE.NOTOP_READY) 		OR 
	(statRef.nSubstate = E_RS_BASE_SUBSTATE.OP_ERROR 		AND 
	 nLastGoodSubstate = E_RS_BASE_SUBSTATE.OP_MONITORING)			THEN
	ActivityMonitoring(TRUE);
ELSIF statRef.nSubstate = E_RS_BASE_SUBSTATE.OP_MONITORING_USER THEN
	ActivityMonitoringUser(TRUE);
ELSIF statRef.nSubstate = E_RS_BASE_SUBSTATE.NOTOP_INITIALIZING THEN
	ActivityInitializing(TRUE);
END_IF

// Set last known good substate. Used for recovery from comm problems.
M_SetLastGoodSubstate();

(* 
	Evaluate state machine transitions.
*)

CASE statRef.nState OF

//***********************************
// NOTOP
//***********************************
E_RS_BASE_STATE.NOTOP:

	(* Transitions from NOTOP substates *)
	CASE statRef.nSubstate OF
	
	E_RS_BASE_SUBSTATE.NOTOP_NOTREADY:		
		IF 	nEvent = E_SM_EVENT.INIT OR cfgRef.bAutoMonitor  THEN
			nEvent := E_SM_EVENT.INIT;
			ActionInitExecute();
			SetState(E_RS_BASE_STATE.NOTOP, E_RS_BASE_SUBSTATE.NOTOP_INITIALIZING);
			SetStatus(E_SM_ERROR.OK, 'OK');
			RETURN;
		END_IF
		
	E_RS_BASE_SUBSTATE.NOTOP_INITIALIZING:			
		IF nEvent = E_SM_EVENT.INITDONE THEN
			nReadType := E_RS_BASE_READ_TYPE.PERIODIC;
			ActivityMonitoring(FALSE);	// Reset Monitoring method
			IF cfgRef.bAutoMonitor THEN
				nEvent := E_SM_EVENT.ENABLE;
				statRef.bAutoStarted	:= TRUE;
				SetState(E_RS_BASE_STATE.OP, E_RS_BASE_SUBSTATE.OP_MONITORING);
			ELSE
				SetState(E_RS_BASE_STATE.NOTOP, E_RS_BASE_SUBSTATE.NOTOP_READY);
			END_IF
			RETURN;
		ELSIF nEvent = E_SM_EVENT.ERRINIT THEN
			// INIT failed. Keep re-trying.
			SetState(E_RS_BASE_STATE.NOTOP, E_RS_BASE_SUBSTATE.NOTOP_NOTREADY);
			RETURN;
		END_IF
		
	E_RS_BASE_SUBSTATE.NOTOP_READY:			
		IF nEvent = E_SM_EVENT.ENABLE THEN
			IF cfgRef.bAutoMonitor THEN
				// Monitoring is already in progress.
				// It has to complete the read cycle in a clean way.
				nNextState		:= E_RS_BASE_STATE.OP;					// Next state after STOP	
				nNextSubstate	:= E_RS_BASE_SUBSTATE.OP_MONITORING;	// Next substate after STOP	
				nNextDescription:= 'BUSY';
				nReadType		:= E_RS_BASE_READ_TYPE.PERIODIC;
				RETURN;
			ELSE
				SetState(E_RS_BASE_STATE.OP, E_RS_BASE_SUBSTATE.OP_MONITORING);
				// This call MUST be after SetState()
				ActivityMonitoring(FALSE);	// Reset Monitoring method
			END_IF
		END_IF

	E_RS_BASE_SUBSTATE.NOTOP_ERROR:			
		IF nEvent = E_SM_EVENT.HWOK THEN
			SetState(E_RS_BASE_STATE.NOTOP, E_RS_BASE_SUBSTATE.NOTOP_NOTREADY);
			RETURN;
		ELSIF nEvent = E_SM_EVENT.COMMOK THEN
			SetState(E_RS_BASE_STATE.NOTOP, nLastGoodSubstate);
			RETURN;			
		END_IF
		
	END_CASE

	(* Transitions from NOTOP state *)
	IF	nEvent = E_SM_EVENT.ERRHW OR
		nEvent = E_SM_EVENT.ERRCOMM	THEN
		ActionUnexpExecute();
		SetState(E_RS_BASE_STATE.NOTOP, E_RS_BASE_SUBSTATE.NOTOP_ERROR);
		RETURN;
	END_IF
	
//***********************************
// OPERATIONAL
//***********************************
E_RS_BASE_STATE.OP:

	(* Transitions from OP subastates *)
	CASE statRef.nSubstate OF
	E_RS_BASE_SUBSTATE.OP_ERROR:			
		IF 	cfgRef.bAutoMonitor  THEN
			nEvent := E_SM_EVENT.INIT;
			ActionInitExecute();
			SetState(E_RS_BASE_STATE.NOTOP, E_RS_BASE_SUBSTATE.NOTOP_INITIALIZING);
			SetStatus(E_SM_ERROR.OK, 'Recovering from error...');
			RETURN;
		END_IF
		IF nEvent = E_SM_EVENT.HWOK THEN
			SetStatus(E_SM_ERROR.OK, 'OK');
			SetState(E_RS_BASE_STATE.OP, E_RS_BASE_SUBSTATE.OP_IDLE);
			RETURN;			
		ELSIF nEvent = E_SM_EVENT.DISABLE THEN
			ActionDisableExecute();
			SetState(E_RS_BASE_STATE.NOTOP, E_RS_BASE_SUBSTATE.NOTOP_ERROR);
			RETURN;			
		ELSIF nEvent = E_SM_EVENT.COMMOK THEN
			SetState(E_RS_BASE_STATE.OP, nLastGoodSubstate);
			RETURN;			
		END_IF

	E_RS_BASE_SUBSTATE.OP_MONITORING:
		IF nEvent = E_SM_EVENT.DISABLE THEN
			ActionDisableExecute();
			RETURN;			
		ELSIF nEvent = E_SM_EVENT.STOPMON THEN
			ActionStopExecute();
			RETURN;			
		ELSIF nEvent = E_SM_EVENT.READDONE THEN
			SetState(E_RS_BASE_STATE.OP, E_RS_BASE_SUBSTATE.OP_IDLE);
			RETURN;			
		ELSIF nEvent = E_SM_EVENT.ERRCOMM THEN
			SetState(E_RS_BASE_STATE.OP, E_RS_BASE_SUBSTATE.OP_ERROR);
			RETURN;			
		END_IF
		
	E_RS_BASE_SUBSTATE.OP_MONITORING_USER:			
		IF nEvent = E_SM_EVENT.DISABLE THEN
			ActionDisableExecute();
			RETURN;			
		ELSIF nEvent = E_SM_EVENT.STOPMON THEN
			ActionStopExecute();
			RETURN;			
		ELSIF nEvent = E_SM_EVENT.READDONE THEN
			SetState(E_RS_BASE_STATE.OP, E_RS_BASE_SUBSTATE.OP_IDLE);
			RETURN;			
		END_IF
		
	E_RS_BASE_SUBSTATE.OP_IDLE:			
		IF nEvent = E_SM_EVENT.DISABLE THEN
			ActionDisableExecute();
			RETURN;			
		ELSIF nEvent = E_SM_EVENT.READ THEN
			nReadType	:= E_RS_BASE_READ_TYPE.SINGLE;
			ActivityMonitoring(FALSE);	// Reset Monitoring method
			SetState(E_RS_BASE_STATE.OP, E_RS_BASE_SUBSTATE.OP_MONITORING);
			RETURN;			
		ELSIF nEvent = E_SM_EVENT.READ_USER THEN
			nReadType	:= E_RS_BASE_READ_TYPE.SINGLE_USER;
			ActivityMonitoringUser(FALSE);	// Reset Monitoring method
			SetState(E_RS_BASE_STATE.OP, E_RS_BASE_SUBSTATE.OP_MONITORING_USER);
			RETURN;			
		ELSIF nEvent = E_SM_EVENT.MONITOR OR nEvent = E_SM_EVENT.ENABLE THEN
			nReadType	:= E_RS_BASE_READ_TYPE.PERIODIC;
			ActivityMonitoring(FALSE);	// Reset Monitoring method
			SetState(E_RS_BASE_STATE.OP, E_RS_BASE_SUBSTATE.OP_MONITORING);
			RETURN;			
		ELSIF nEvent = E_SM_EVENT.MONITOR_USER THEN
			nReadType	:= E_RS_BASE_READ_TYPE.PERIODIC_USER;
			ActivityMonitoringUser(FALSE);	// Reset Monitoring method
			SetState(E_RS_BASE_STATE.OP, E_RS_BASE_SUBSTATE.OP_MONITORING_USER);
			RETURN;			
		END_IF
		
	END_CASE
	
	// Transitions from OP state.
	// Valid for any OP substate.
	IF nEvent = E_SM_EVENT.ERRHW THEN
		ActionUnexpExecute();
		SetState(E_RS_BASE_STATE.OP, E_RS_BASE_SUBSTATE.OP_ERROR);
		RETURN;
	ELSIF nEvent = E_SM_EVENT.ERRCOMM THEN
		SetState(E_RS_BASE_STATE.OP, E_RS_BASE_SUBSTATE.OP_ERROR);
		RETURN;
	END_IF
	
END_CASE

(* 
	"Global" internal transitions valid in any state should go here.
	They do not change the active state configuration. 
	They are evaluated after all the others transitions have been 
	considered.
*) 
IF nEvent = E_SM_EVENT.RESET THEN
	ActionResetExecute();
	SetState(E_RS_BASE_STATE.NOTOP, E_RS_BASE_SUBSTATE.NOTOP_NOTREADY);
	RETURN;
END_IF
END_METHOD

END_FUNCTION_BLOCK

// ---- POUs/Coolers/FB_RS_COMM_CRYOTELGT.TcPOU
FUNCTION_BLOCK FB_RS_COMM_CRYOTELGT EXTENDS FB_RS_COMM_BASE
VAR_INPUT
END_VAR
VAR_OUTPUT
END_VAR
VAR CONSTANT
END_VAR
VAR
	{attribute 'OPC.UA.DA' := '1'}
	cfg:		T_RS_COMM_CFG;				// Config parameters
	{attribute 'OPC.UA.DA' := '1'}
	ctrl:		T_RS_COMM_CTRL;				// Control parameters
	{attribute 'OPC.UA.DA' := '1'}
	{attribute 'OPC.UA.DA.Access' := '1'}
	info:		T_RS_COMM_INFO; 			// Info parameters - ReadOnly
	{attribute 'OPC.UA.DA' := '1'}
	{attribute 'OPC.UA.DA.Access' := '1'}
	stat:		T_RS_COMM_STAT;				// Status parameters - ReadOnly

	sim:		FB_SIM_RS_COMM_CRYOTELGT;		// COMM simulator

	// Physical signals - to be mapped to EL60xx serial port controller !!!
	COMin_EL60xx	AT %I* 	: KL6inData22B;	(* linked to the EL60xx *)
	COMout_EL60xx	AT %Q*	: KL6outData22B;(* linked to the EL60xx *)

	(* Serial line control *)
	COMportControl: 		SerialLineControl;

END_VAR

// Set references
cfgRef	REF=cfg;
ctrlRef	REF=ctrl;
infoRef	REF=info;
statRef	REF=stat;
simRef	REF=sim;

SUPER^();

METHOD M_ActionInitExecute
VAR_INPUT
END_VAR
//
// Copy input parameters to cfg
//
cfg.sCmdSuffix		:= in_sCmdSuffix;
cfg.sReplySuffix	:= in_sReplySuffix;
cfg.nTimeout		:= in_nTimeout;

//
// If in simulation, there is no need to reset anything.
// Just set it to initialised and go to IDLE state.
//
IF in_bSimulation THEN
	fbTimer (IN := FALSE);
	statRef.bInitialised	:= TRUE;
	statRef.nStatus			:= E_RS_COMM_STATUS.IDLE;
	statRef.sStatus			:= 'INITIALISED';
	State 					:= E_RS_COMM_STATE.IDLE;
ELSE
	stat.bInitialised	:= FALSE;
	stat.sStatus		:= 'INITIALISING';
	stat.nStatus		:= E_RS_COMM_STATUS.BUSY;
	stat.sReply 		:= ''; (* No reply yet *)
	stat.nErrorCode		:= E_RS_COMM_ERROR.OK;
	stat.sErrorText		:= 'OK';
	
	// Reset the connected serial hardware 
	ComReset (
		Execute 	:= FALSE,
		pComIn		:= ADR(COMin_EL60xx),
		pComOut		:= ADR(COMout_EL60xx),
		SizeComIn	:= SIZEOF(COMin_EL60xx),
		);
	
	// Set next state
	State 	:= E_RS_COMM_STATE.RESET;
END_IF
END_METHOD

METHOD M_ComPortControl
VAR_INPUT
END_VAR
// RS specific call of the background communication process
COMportControl(
	Mode		:= ComSerialLineMode_t.SERIALLINEMODE_KL6_22B_STANDARD,
	pComIn		:= ADR(COMin_EL60xx),					(* I/O data; see global variables *)
	pComOut		:= ADR(COMout_EL60xx),					(* I/O data; see global variables *)
	SizeComIn	:= UINT_TO_INT(SIZEOF(COMin_EL60xx)),	(* I/O data; see global variables *)
	TxBuffer	:= TxBuffer,							(* transmit buffer; see global variables *)
	RxBuffer	:= RxBuffer);							(* receive buffer; see global variables *)
END_METHOD

METHOD M_Reset
VAR_INPUT
END_VAR
// RS specific call of communication reset
//
// Reset the connected serial hardware.
ComReset (
	Execute 	:= TRUE,
	pComIn		:= ADR(COMin_EL60xx),
	pComOut		:= ADR(COMout_EL60xx),
	SizeComIn	:= SIZEOF(COMin_EL60xx),
	);

(* Next step is to clear the buffers *)
IF ComReset.Done THEN
	fbTimer (IN := FALSE);	// Reset the timer
	State 		:= E_RS_COMM_STATE.CLEAR_BUFFER;
END_IF
END_METHOD

END_FUNCTION_BLOCK

